	{attribute 'TcHmiSymbol.Show'}

	bSimulated:		BOOL;				// Flag indicating if the value is simulated.
	{attribute 'TcHmiSymbol.Show'}

	lrSimTempK:	LREAL;				// Simulated Temp [K]

	{attribute 'TcHmiSymbol.Show'}

	bEnabled:		BOOL	:= FALSE;	// Flag indicating if the voter is enabled
    
	{attribute 'TcHmiSymbol.Show'}

	sDescription:	STRING;	// User description of the voter (e.g. 'Average detector T')
    
	{attribute 'TcHmiSymbol.Show'}

	bValid:			BOOL	:= FALSE;	// Flag indicating if the value is valid.
	{attribute 'TcHmiSymbol.Show'}
	{attribute 'TcHmiSymbol.ReadOnly'}
	lrTempK:		LREAL;				// Calculated Temperature in K
	sStatus:		STRING;				// Status string

	// Flags indicating connected sensor is Valid.
	{attribute 'TcHmiSymbol.Show'}
	{attribute 'TcHmiSymbol.ReadOnly'}
	lrSens1TempK:		LREAL;
	{attribute 'TcHmiSymbol.Show'}
	{attribute 'TcHmiSymbol.ReadOnly'}
	lrSens2TempK:		LREAL;
	{attribute 'TcHmiSymbol.Show'}
	{attribute 'TcHmiSymbol.ReadOnly'}
	lrSens3TempK:		LREAL;
	{attribute 'TcHmiSymbol.Show'}
	{attribute 'TcHmiSymbol.ReadOnly'}
	lrSens4TempK:		LREAL;
	{attribute 'TcHmiSymbol.Show'}
	{attribute 'TcHmiSymbol.ReadOnly'}
	lrSens5TempK:		LREAL;
	
	{attribute 'TcHmiSymbol.Show'}
	{attribute 'TcHmiSymbol.ReadOnly'}
	bValidSensor1:		BOOL	:= FALSE;
	{attribute 'TcHmiSymbol.Show'}
	{attribute 'TcHmiSymbol.ReadOnly'}
	bValidSensor2:		BOOL	:= FALSE;
	{attribute 'TcHmiSymbol.Show'}
	{attribute 'TcHmiSymbol.ReadOnly'}
	bValidSensor3:		BOOL	:= FALSE;
	{attribute 'TcHmiSymbol.Show'}
	{attribute 'TcHmiSymbol.ReadOnly'}
	bValidSensor4:		BOOL	:= FALSE;
	{attribute 'TcHmiSymbol.Show'}
	{attribute 'TcHmiSymbol.ReadOnly'}
	bValidSensor5:		BOOL	:= FALSE;
	{attribute 'TcHmiSymbol.ShowRecursively'}

	stAlarms:		T_CRYO_ALARMS;	

	bInRange:		BOOL	:= FALSE;

	lrTempC:		LREAL;				// Temp [deg C]
	
	{attribute 'TcHmiSymbol.Show'}
	aTempIndexes:		ARRAY[0..4] OF E_ALL_METIS_TEMPERATURES;
	{attribute 'TcHmiSymbol.Show'}
	nVoteMethod:		E_METIS_TEMP_VOTE_METHOD;

    //bEnabled:       BOOL;	

END_STRUCT
END_TYPE

// DUTs/Structures/Temp_Voter/T_METIS_TEMP_VOTE_CFG
TYPE T_METIS_TEMP_VOTE_CFG :
STRUCT
    bEnabled        : BOOL;
    sDescription    : STRING; 

	sTemp1_Name	    : STRING;
	sTemp2_Name	    : STRING;
	sTemp3_Name	    : STRING;
	sTemp4_Name	    : STRING;
	sTemp5_Name	    : STRING;
	
	nVote_Method    : E_METIS_TEMP_VOTE_METHOD;
	
	eTemperature1   : E_ALL_METIS_TEMPERATURES;
	eTemperature2   : E_ALL_METIS_TEMPERATURES;
	eTemperature3   : E_ALL_METIS_TEMPERATURES;
	eTemperature4   : E_ALL_METIS_TEMPERATURES;
	eTemperature5   : E_ALL_METIS_TEMPERATURES;
	
END_STRUCT
END_TYPE

// DUTs/Structures/Temp_Voter/T_METIS_TEMP_VOTERS_CTRL
TYPE T_METIS_TEMP_VOTERS_CTRL :
STRUCT
	
	// CRY

    tor_vote_cry_1  :			FB_CRYO_CMD_OVERRIDE;
    tor_vote_cry_2  :           FB_CRYO_CMD_OVERRIDE;
    tor_vote_cry_3  :           FB_CRYO_CMD_OVERRIDE;
    tor_vote_cry_4  :           FB_CRYO_CMD_OVERRIDE;
    tor_vote_cry_5  :           FB_CRYO_CMD_OVERRIDE;
    tor_vote_cry_6  :           FB_CRYO_CMD_OVERRIDE;
    tor_vote_cry_7  :           FB_CRYO_CMD_OVERRIDE;
    tor_vote_cry_8  :           FB_CRYO_CMD_OVERRIDE;
    tor_vote_cry_9  :           FB_CRYO_CMD_OVERRIDE;
    tor_vote_cry_10 :           FB_CRYO_CMD_OVERRIDE;
                                
    // SCA                      
    tor_vote_sca_1  :           FB_CRYO_CMD_OVERRIDE;
    tor_vote_sca_2  :           FB_CRYO_CMD_OVERRIDE;
    tor_vote_sca_3  :           FB_CRYO_CMD_OVERRIDE;
    tor_vote_sca_4  :           FB_CRYO_CMD_OVERRIDE;
    tor_vote_sca_5  :           FB_CRYO_CMD_OVERRIDE;
    tor_vote_sca_6  :           FB_CRYO_CMD_OVERRIDE;
    tor_vote_sca_7  :           FB_CRYO_CMD_OVERRIDE;
    tor_vote_sca_8  :           FB_CRYO_CMD_OVERRIDE;
    tor_vote_sca_9  :           FB_CRYO_CMD_OVERRIDE;
    tor_vote_sca_10 :           FB_CRYO_CMD_OVERRIDE;
                                
    // IMG                      
    tor_vote_img_1  :           FB_CRYO_CMD_OVERRIDE;
    tor_vote_img_2  :           FB_CRYO_CMD_OVERRIDE;
    tor_vote_img_3  :           FB_CRYO_CMD_OVERRIDE;
    tor_vote_img_4  :           FB_CRYO_CMD_OVERRIDE;
    tor_vote_img_5  :           FB_CRYO_CMD_OVERRIDE;
    tor_vote_img_6  :           FB_CRYO_CMD_OVERRIDE;
    tor_vote_img_7  :           FB_CRYO_CMD_OVERRIDE;
    tor_vote_img_8  :           FB_CRYO_CMD_OVERRIDE;
    tor_vote_img_9  :           FB_CRYO_CMD_OVERRIDE;
    tor_vote_img_10 :           FB_CRYO_CMD_OVERRIDE;
                                
    // System temp               
    tor_vote_master_temp:       FB_CRYO_CMD_OVERRIDE;
    tor_vote_master_1   :       FB_CRYO_CMD_OVERRIDE;
    tor_vote_master_2   :       FB_CRYO_CMD_OVERRIDE;
	
	
// Temp Simulation Flag

	//CRY
	bSim_Temp_vote_cry_1  :		BOOL := FALSE;
    bSim_Temp_vote_cry_2  :     BOOL := FALSE;
    bSim_Temp_vote_cry_3  :     BOOL := FALSE;
    bSim_Temp_vote_cry_4  :     BOOL := FALSE;
    bSim_Temp_vote_cry_5  :     BOOL := FALSE;
    bSim_Temp_vote_cry_6  :     BOOL := FALSE;
    bSim_Temp_vote_cry_7  :     BOOL := FALSE;
    bSim_Temp_vote_cry_8  :     BOOL := FALSE;
    bSim_Temp_vote_cry_9  :     BOOL := FALSE;
    bSim_Temp_vote_cry_10 :     BOOL := FALSE;
                                
    //SCA                       
    bSim_Temp_vote_sca_1  :     BOOL := FALSE;
    bSim_Temp_vote_sca_2  :     BOOL := FALSE;
    bSim_Temp_vote_sca_3  :     BOOL := FALSE;
    bSim_Temp_vote_sca_4  :     BOOL := FALSE;
    bSim_Temp_vote_sca_5  :     BOOL := FALSE;
    bSim_Temp_vote_sca_6  :     BOOL := FALSE;
    bSim_Temp_vote_sca_7  :     BOOL := FALSE;
    bSim_Temp_vote_sca_8  :     BOOL := FALSE;
    bSim_Temp_vote_sca_9  :     BOOL := FALSE;
    bSim_Temp_vote_sca_10 :     BOOL := FALSE;
                                
	//IMG                       
    bSim_Temp_vote_img_1  :     BOOL := FALSE;
    bSim_Temp_vote_img_2  :     BOOL := FALSE;
    bSim_Temp_vote_img_3  :     BOOL := FALSE;
    bSim_Temp_vote_img_4  :     BOOL := FALSE;
    bSim_Temp_vote_img_5  :     BOOL := FALSE;
    bSim_Temp_vote_img_6  :     BOOL := FALSE;
    bSim_Temp_vote_img_7  :     BOOL := FALSE;
    bSim_Temp_vote_img_8  :     BOOL := FALSE;
    bSim_Temp_vote_img_9  :     BOOL := FALSE;
    bSim_Temp_vote_img_10 :     BOOL := FALSE;
                                
    //system temp               
    bSim_Temp_vote_master_temp: BOOL := FALSE;
    bSim_Temp_vote_master_1   : BOOL := FALSE;
    bSim_Temp_vote_master_2   : BOOL := FALSE;
                             
	
                               
END_STRUCT
END_TYPE

// DUTs/Structures/Temperature/E_ALL_METIS_TEMPERATURES
{attribute 'qualified_only'}
{attribute 'strict'}
{attribute 'to_string'}
TYPE E_ALL_METIS_TEMPERATURES :
(
	empty_temp 		:= 0,					
	(*Temp Cryo: 23 + 10 = 33 *)
	t_cry_sha_1		:= 1,			
	t_cry_sha_2		:= 2,			
	t_cry_sha_3		:= 3,			
	t_cry_sha_4		:= 4,           	
	t_cry_shb_1		:= 5,			
	t_cry_shb_2		:= 6,           	
	t_cry_shb_3		:= 7,           	
	t_cry_shb_4		:= 8,           	
	t_cry_shc_1		:= 9,			
	t_cry_shc_2		:= 10,           	
	t_cry_shc_3     := 11,           	
	t_cry_shc_4     := 12,           	
	t_cry_pta_1     := 13,           	
	t_cry_pta_2     := 14,           	
	t_cry_ptb_1     := 15,           	
	t_cry_ptb_2     := 16,           	
	t_cry_ptc_1		:= 17,			
	t_cry_ptc_2     := 18,           	
	t_cry_pta_3     := 19,           	
	t_cry_ptb_3     := 20,           	
	t_cry_ptc_3     := 21,           	
	t_cry_sp_1		:= 22,			
	t_cry_sp_2		:= 23,			
	// voter outputs (10)           
	t_cry_vot_1     := 24,            
	t_cry_vot_2     := 25,            
	t_cry_vot_3     := 26,            
	t_cry_vot_4     := 27,            
	t_cry_vot_5     := 28,            
	t_cry_vot_6     := 29,            
	t_cry_vot_7     := 30,            
	t_cry_vot_8     := 31,            
	t_cry_vot_9     := 32,            
	t_cry_vot_10    := 33,            
	                            
	(*SCA Temps: 16 + 4 + 10 + 3 = 33 *)  
	         
	// cu X2
	t_sca_fw_1       := 34,           
	t_sca_fw_2       := 35,           
	t_sca_lu_1       := 36,           
	t_sca_fm         := 37,           
	t_sca_fs         := 38,           
	t_sca_lu_2       := 39,           
	t_sca_mod        := 40,           
	t_sca_pyr		 := 41,		
	// cu X3                    
	t_sca_h_1        := 42,           
	t_sca_if_1       := 43,           
	t_sca_if_2       := 44,           
	t_sca_lu_3       := 45,           
	t_sca_bp_1       := 46,           
	t_sca_bp_2       := 47,           
	t_sca_bp_3       := 48,           
	t_sca_h_2        := 49,           
	// detector (4)             
	t_sca_det_1      := 50,           
	t_sca_det_2      := 51,           
	t_sca_dhs_1      := 52,           
	t_sca_dhs_2      := 53,           
// voter outputs(10)        
	t_sca_vot_1       := 54,          
	t_sca_vot_2       := 55,          
	t_sca_vot_3       := 56,          
	t_sca_vot_4       := 57,          
	t_sca_vot_5       := 58,          
	t_sca_vot_6       := 59,          
	t_sca_vot_7       := 60,          
	t_sca_vot_8       := 61,          
	t_sca_vot_9       := 62,          
	t_sca_vot_10      := 63,          
	// temperature controller ramps (3)
	t_sca_wuh_ramp    := 64,         
	t_sca_det_2_ramp  := 65,         
	t_sca_dhs_2_ramp  := 66,         
	
	(*IMG Temps : 24 + 6 + 10 + 4 = 44 *)              
	
	// cu (24)			  
	t_img_lpw_1        := 67,        
	t_img_lpw_2        := 68,         
	t_img_lfw_1        := 69,         
	t_img_lfw_2        := 70,         
	t_img_lpr_1        := 71,         
	t_img_bwu_3        := 72,         
	t_img_lnd_1        := 73,         
	t_img_lnd_2        := 74,         
	t_img_npw_1        := 75,         
	t_img_npw_2        := 76,         
	t_img_nfw_1        := 77,         
	t_img_nfw_2        := 78,         
	t_img_npr_1        := 79,         
	t_img_bwu_2        := 80,         
	t_img_nnd_1        := 81,         
	t_img_nnd_2        := 82,         
	t_img_opt_1        := 83,         
	t_img_bwu_1        := 84,         
	t_img_ctr_1        := 85,         
	t_img_ctr_2        := 86,         
	t_img_70k_1        := 87,         
	t_img_ln2_1        := 88,         
	t_img_ln2_2		   := 89,    
	t_img_hex_1        := 90,         
	// detector (6)             
	t_img_lmd_1        := 91,         
	t_img_lmd_2        := 92,         
	t_img_lmp_1        := 93,         
	t_img_lmp_2        := 94,         
	t_img_nd_1         := 95,         
	t_img_nd_2         := 96,         
	// voter outputs (10) 
	t_img_vot_1        := 97,      
	t_img_vot_2        := 98,        
	t_img_vot_3        := 99,       
	t_img_vot_4        := 100,       
	t_img_vot_5        := 101,       
	t_img_vot_6        := 102,       
	t_img_vot_7        := 103,       
	t_img_vot_8        := 104,       
	t_img_vot_9        := 105,       
	t_img_vot_10       := 106,       
// temperature controller       ramps (4)
	t_img_wuh_ramp     := 107,       
	t_img_lmd_2_ramp   := 108,       
	t_img_lmp_2_ramp   := 109,       
	t_img_nd_2_ramp    := 110,       
	                            
	(*Temp LMS : 16 *)          
	                            
	t_lms_pma_1        := 111,         
	t_lms_pma_2        := 112,         
	t_lms_msa_1        := 113,         
	t_lms_msa_2        := 114,         
	t_lms_pra_1        := 115,         
	t_lms_pra_2        := 116,         
	t_lms_gra_1        := 117,         
	t_lms_gra_2        := 118,         
	t_lms_pla_1        := 119,         
	t_lms_pla_2        := 120,         
	t_lms_pla_3        := 121,         
	t_lms_pla_4        := 122,         
	t_lms_tma          := 123,         
	t_lms_dtw          := 124,         
	t_lms_ptw          := 125,         
	t_lms_spare        := 126,         
	                            
	(*Temp CFO*) 
	
	
	// RTD temperatures   
	t_cry_pca          := 127,          // PCA.T = IMG Heat Exchanger Out
	t_cry_pcb          := 128,          // PCB.T = CFO Heat Exchanger Out
	t_cry_wim          := 129,          // WI.MT = Window Mount
	t_cry_wia          := 130,          // WI.AT = Window Ambient
                          
	// dew point temperatures
	t_cry_wid          := 131,         
	
	(*System temperatures   (3) *)
	// Master temperature to estimate overall temperature of the cryostat  
						  
	t_master           := 132,      	
	t_master_vot_1     := 133,      	
	t_master_vot_2     := 134     	
	                      

	
);
END_TYPE

// DUTs/Structures/Temperature/T_METIS_TEMPERATURE_STATUS
TYPE T_METIS_TEMPERATURE_STATUS EXTENDS T_METIS_SENSOR_BASE_STATUS:
STRUCT
	{attribute 'TcHmiSymbol.Show'}
    lrTempC : LREAL;
	{attribute 'TcHmiSymbol.Show'}
    lrTempK : LREAL;
END_STRUCT
END_TYPE

// HMI/DUTs/Cryo_Devices/Temperatures/E_HMI_TEMP_TABS
{attribute 'qualified_only'}
{attribute 'strict'}
TYPE E_HMI_TEMP_TABS :
(
    VOTERS
);
END_TYPE

// HMI/DUTs/Cryo_Devices/E_HMI_PUMPS_TABS
{attribute 'qualified_only'}
{attribute 'strict'}
TYPE E_HMI_PUMPS_TABS :
(
	RP_BRANCH_A := 0,
	TP_BRANCH_A,
	RP_BRANCH_B,
	TP_BRANCH_B
);
END_TYPE

// HMI/DUTs/Subsystems/CFO/E_HMI_CFO_TABS
{attribute 'qualified_only'}
{attribute 'strict'}
TYPE E_HMI_CFO_TABS :
(
	TEMPERATURES,
    VOTERS,
    HEATERS,
    TCONTROL
);
END_TYPE

// HMI/DUTs/Subsystems/CRY/Components/E_HMI_CRY_HEATER_TABS
{attribute 'qualified_only'}
{attribute 'strict'}
TYPE E_HMI_CRY_HEATER_TABS :
(
    H_CRY_SHA,
    H_CRY_SHB,
    H_CRY_SHC,
    H_CRY_SP,
    H_CRY_PTA,
    H_CRY_PTB,
    H_CRY_PTC,
    H_CRY_WI
);
END_TYPE

// HMI/DUTs/Subsystems/CRY/Components/E_HMI_CRY_TC_TABS
{attribute 'qualified_only'}
{attribute 'strict'}
TYPE E_HMI_CRY_TC_TABS :
(
	TC_CRY_SHA,
    TC_CRY_SHB,
    TC_CRY_SHC,
    TC_CRY_PT,
    TC_CRY_WI,
	TC_CRY_SP
);
END_TYPE

// HMI/DUTs/Subsystems/CRY/E_HMI_CRY_TABS
{attribute 'qualified_only'}
{attribute 'strict'}
TYPE E_HMI_CRY_TABS :
(
	TEMPERATURES,
    RH,
    HEATERS,
    VOTERS,
    TCONTROL,
	LN2CONTROL
);
END_TYPE

// HMI/DUTs/Subsystems/ICS/E_HMI_ICS_TABS
{attribute 'qualified_only'}
{attribute 'strict'}
TYPE E_HMI_ICS_TABS :
(
	CCU_NS_1,
	CCU_NS_2,
	CCU_CONFIGS
);
END_TYPE

// HMI/DUTs/Subsystems/IMG/Components/E_HMI_IMG_HEATER_TABS
{attribute 'qualified_only'}
{attribute 'strict'}
TYPE E_HMI_IMG_HEATER_TABS :
(
	H_IMG_WUH_1,
    H_IMG_WUH_2,
    H_IMG_LMD_2,
    H_IMG_LMP_2,
    H_IMG_ND_2
);
END_TYPE

// HMI/DUTs/Subsystems/IMG/Components/E_HMI_IMG_TC_TABS
{attribute 'qualified_only'}
{attribute 'strict'}
TYPE E_HMI_IMG_TC_TABS :
(
	TC_IMG_WUH,
    TC_IMG_LMD_2,
    TC_IMG_LMP_2,
    TC_IMG_ND_2
);
END_TYPE

// HMI/DUTs/Subsystems/IMG/E_HMI_IMG_TABS
{attribute 'qualified_only'}
{attribute 'strict'}
TYPE E_HMI_IMG_TABS :
(
	TEMPERATURES,
    VOTERS,
    TCONTROL,
    HEATERS,
    LAKESHORE_LM_DET,
    LAKESHORE_N_DET
);
END_TYPE

// HMI/DUTs/Subsystems/LMS/E_HMI_LMS_TABS
{attribute 'qualified_only'}
{attribute 'strict'}
TYPE E_HMI_LMS_TABS :
(
	TEMPERATURES,
    VOTERS,
    HEATERS,
    TCONTROL
);
END_TYPE

// HMI/DUTs/Subsystems/SCA/Components/E_HMI_SCA_HEATER_TABS
{attribute 'qualified_only'}
{attribute 'strict'}
TYPE E_HMI_SCA_HEATER_TABS :
(
	H_SCA_WUH_1,
    H_SCA_WUH_2,
    H_SCA_DET_2,
    H_SCA_DHS_2
);
END_TYPE

// HMI/DUTs/Subsystems/SCA/Components/E_HMI_SCA_TC_TABS
{attribute 'qualified_only'}
{attribute 'strict'}
TYPE E_HMI_SCA_TC_TABS :
(
	TC_SCA_WUH,
    TC_SCA_DET_2,
    TC_SCA_DHS_2
);
END_TYPE

// HMI/DUTs/Subsystems/SCA/E_HMI_SCA_TABS
{attribute 'qualified_only'}
{attribute 'strict'}
TYPE E_HMI_SCA_TABS :
(
	TEMPERATURES,
    VOTERS,
    TCONTROL,
    HEATERS,
    LAKESHORE_DET
);
END_TYPE

// HMI/DUTs/System/E_HMI_TABS
{attribute 'qualified_only'}
{attribute 'strict'}
TYPE E_HMI_TABS :
(
	HOME,
    SERVICES,
	EVACUATION,
    COOL_DOWN,
	WARM_UP,
	VENTING,
	ANTI_FOGGING,
	REGENERATION,
	POWER_OUTAGE,
	CABINETS,
	VALVES,
	CONTROL_UNITS,
	SUBSYSTEMS_CRY,
    SUBSYSTEMS_CFO,
    SUBSYSTEMS_IMG,
    SUBSYSTEMS_LMS,
    SUBSYSTEMS_SCA,
    SUBSYSTEMS_ICS,
	HEATERS,
	EVENTS,
	PRESSURES,
	COOLERS,
	PUMPS,
	TEMPERATURES,
	ICS_INTERLOCKS,
	DETECTORS,
	CONTROL_LOOPS,
	SIMULATION
	
);
END_TYPE

// HMI/DUTs/Util/E_HMI_COLORS
TYPE E_HMI_COLORS :
(
	GREEN := 16#FF00FF00,
	RED := 16#FFFF0000,
	ORANGE := 16#FFFF802D,
	GRAY := 16#FFD3D3D3,
	DARK_GRAY := 16#FF949494,
	BLACK := 16#FF000000,
	WHITE := 16#FFFFFFFF,
	BLUE := 16#FF0000FF
) DWORD;
END_TYPE

// HMI/DUTs/Util/E_HMI_VOTER_TABS
{attribute 'qualified_only'}
{attribute 'strict'}
TYPE E_HMI_VOTER_TABS :
(
	VOTER_1,
    VOTER_2,
    VOTER_3,
    VOTER_4,
    VOTER_5,
    VOTER_6,
    VOTER_7,
    VOTER_8,
    VOTER_9,
    VOTER_10
);
END_TYPE

// HMI/DUTs/Util/T_ECAT_MODULE
TYPE T_ECAT_MODULE :
STRUCT
    sName : STRING(32);
    sType : STRING(16);
    nState : UINT;
    sState : STRING(16);
    bError : BOOL;
    bDisabled : BOOL;
    bNotPresent : BOOL;
END_STRUCT
END_TYPE

// HMI/DUTs/Util/T_HMI_COLORS
TYPE T_HMI_COLORS :
STRUCT
    fg : E_HMI_COLORS; // foreground
    bg : E_HMI_COLORS; // background
END_STRUCT
END_TYPE

// POUs/Devices/DigitalOutput/T_METIS_DO_CTRL
TYPE T_METIS_DO_CTRL :
STRUCT
    bEnable : BOOL;
END_STRUCT
END_TYPE

// POUs/Devices/DigitalOutput/T_METIS_DO_STAT
TYPE T_METIS_DO_STAT :
STRUCT    
    bActive             : BOOL; // Actual output (TRUE = Active, FALSE = Inactie)
    
    bError              : BOOL; // summary of the fault flags
    
	bOvertemperature    : BOOL; // Over temperature fault
	bOpenLoad           : BOOL; // Open load fault
	bOverCurrent        : BOOL; // Over current fault
	bShortCircuit       : BOOL; // Short circuit fault
    
    sStatus             : STRING;
END_STRUCT
END_TYPE

// POUs/Devices/RH_Sensor/T_METIS_RH_SENSOR_STAT
TYPE T_METIS_RH_SENSOR_STAT EXTENDS T_CRYO_SENSOR_STATUS:
STRUCT
    lrRhFraction        : LREAL; // Relative Humidity as a fraction [0..1]
    lrRhPercent         : LREAL; // Relative Humidity as a percentage [0..100]
    lrDewPointTempC     : LREAL; // Dew point temperature in °C
    bDewPointTempValid  : BOOL;  // TRUE if the dew point is valid
END_STRUCT
END_TYPE

// HMI/POUs/Cryo-Routines/Anti-Fogging/FB_HMI_ANTI_FOGGING
FUNCTION_BLOCK FB_HMI_ANTI_FOGGING EXTENDS FB_HMI_COMPONENT
VAR_INPUT
END_VAR
VAR_OUTPUT
END_VAR
VAR
END_VAR
VAR_IN_OUT
	{attribute 'OPC.UA.DA' := '0'}
	fbInstance		: FB_METIS_CRYO_ANTI_FOGGING;
	{attribute 'OPC.UA.DA' := '0'}
	interlocks:						T_METIS_CRYO_INTERLOCKS;

END_VAR


fbHealthStatus( 
				bIsEnabled:= TRUE, 
				bIsGood := NOT fbInstance.stat.bError,
				bHasWarning := fbInstance.stat.bWarning OR interlocks.bInterlock_AntiFogging
				);
				
fbBusyStatus(
				bIsBusy := fbInstance.stat.bBusy,
				bIsEnabled := TRUE);
				
M_UpdateStatusColor();

END_FUNCTION_BLOCK

// HMI/POUs/Util/Component/FB_HMI_COMPONENT
FUNCTION_BLOCK FB_HMI_COMPONENT
VAR_INPUT
END_VAR
VAR_OUTPUT
    fbHealthStatus : FB_HMI_HEALTH_STATUS;
    fbBusyStatus : FB_HMI_BUSY_STATUS;
    fbStatusColor : T_HMI_COLORS;
END_VAR
VAR
END_VAR

METHOD PROTECTED M_UpdateStatusColor
VAR_INPUT
END_VAR
// health and busy states must be updated by the subtype before calling this method!
fbStatusColor := F_HMI_HEALTH_BUSY_TO_COLOR(fbHealthStatus, fbBusyStatus);
END_METHOD

END_FUNCTION_BLOCK

// HMI/POUs/Services/Status/FB_HMI_HEALTH_STATUS
FUNCTION_BLOCK FB_HMI_HEALTH_STATUS
VAR_INPUT
	// TRUE if the subject is in Good health
	bIsGood: BOOL;
	// TRUE to add a warning to the Good health state
	bHasWarning: BOOL := FALSE;
	// TRUE if the health status is used
	bIsEnabled: BOOL := TRUE;
END_VAR
VAR_OUTPUT
	// TRUE if the subject is enabled
	bEnabled: BOOL;
    // TRUE if the subject is in good health
	bGood: BOOL;
	// TRUE if the subject is in good health, but there are one or more warnings present
	bWarning: BOOL;
	// TRUE if the subject is in bad health
	bBad: BOOL;
END_VAR
VAR_IN_OUT
END_VAR
VAR
END_VAR

bEnabled := bIsEnabled;
bBad := (NOT(bIsGood)) AND bIsEnabled;
bGood := (bIsGood AND (NOT(bHasWarning))) AND bIsEnabled;
bWarning := (bIsGood AND bHasWarning) AND bIsEnabled;

END_FUNCTION_BLOCK

// HMI/POUs/Services/Status/FB_HMI_BUSY_STATUS
FUNCTION_BLOCK FB_HMI_BUSY_STATUS
VAR_INPUT
	// TRUE if busy
	bIsBusy: BOOL;
	// TRUE if the busy status is used
	bIsEnabled: BOOL := TRUE;
END_VAR
VAR_OUTPUT
	// TRUE if the subject is enabled
	bEnabled: BOOL;
	///The subject is idle
	bIdle: BOOL;
	///The subject is busy
	bBusy: BOOL;
END_VAR
VAR_IN_OUT
END_VAR
VAR
END_VAR

bBusy := bIsBusy AND bIsEnabled;
bIdle := (NOT(bIsBusy)) AND bIsEnabled;

END_FUNCTION_BLOCK

// HMI/POUs/Services/Status/F_HMI_HEALTH_BUSY_TO_COLOR
FUNCTION F_HMI_HEALTH_BUSY_TO_COLOR : T_HMI_COLORS
VAR_IN_OUT
    fbHealthStatus : FB_HMI_HEALTH_STATUS;
    fbBusyStatus   : FB_HMI_BUSY_STATUS;
END_VAR
VAR_OUTPUT
END_VAR
VAR
END_VAR

IF fbHealthStatus.bGood THEN
	IF fbBusyStatus.bBusy THEN
		F_HMI_HEALTH_BUSY_TO_COLOR.fg := E_HMI_COLORS.WHITE;
		F_HMI_HEALTH_BUSY_TO_COLOR.bg := E_HMI_COLORS.BLUE;
	ELSE
		F_HMI_HEALTH_BUSY_TO_COLOR.fg := E_HMI_COLORS.BLACK;
		F_HMI_HEALTH_BUSY_TO_COLOR.bg := E_HMI_COLORS.GREEN;
	END_IF
ELSIF fbHealthStatus.bBad THEN
	F_HMI_HEALTH_BUSY_TO_COLOR.fg := E_HMI_COLORS.WHITE;
	F_HMI_HEALTH_BUSY_TO_COLOR.bg := E_HMI_COLORS.RED;
ELSIF fbHealthStatus.bWarning THEN
	F_HMI_HEALTH_BUSY_TO_COLOR.fg := E_HMI_COLORS.WHITE;
	F_HMI_HEALTH_BUSY_TO_COLOR.bg := E_HMI_COLORS.ORANGE;
ELSE
	F_HMI_HEALTH_BUSY_TO_COLOR.fg := E_HMI_COLORS.BLACK;
	F_HMI_HEALTH_BUSY_TO_COLOR.bg := E_HMI_COLORS.GRAY;
END_IF

END_FUNCTION

// POUs/Routines/AntiFogging/FB_METIS_CRYO_ANTI_FOGGING
FUNCTION_BLOCK FB_METIS_CRYO_ANTI_FOGGING
VAR_INPUT
	in_sName:							STRING := 'ANTI-FOGGING';
	in_bEnable:							BOOL := FALSE;
	in_Cryo_Stat:						T_METIS_CRYO_STAT;
	in_lrAntiFog_Purging_DewPoint:		LREAL := 10.0; // If dew-point is <10 K below ambient window purging is started
	in_lrAntiFog_Heating_DewPoint:		LREAL := 10.0; // If dew-point is <5 K below ambient window increased window heating is started
	in_lrAntiFog_DewPoint_Alarm:		LREAL := 5.0;  // dew point is <5 K below window temperature
END_VAR
VAR_OUTPUT
	out_bAntiFoggingActive:			BOOL := FALSE;
END_VAR
VAR_IN_OUT
	{attribute 'OPC.UA.DA' := '0'}
	all_cryo_temps:					FB_METIS_TEMPERATURES;
	{attribute 'OPC.UA.DA' := '0'}
	all_heaters:					FB_METIS_HEATERS;
	{attribute 'OPC.UA.DA' := '0'}
	all_t_ctrls:      				FB_METIS_TCTRL;
	{attribute 'OPC.UA.DA' := '0'}
	all_t_votes: 					FB_METIS_VOTERS;
	{attribute 'OPC.UA.DA' := '0'}
	interlocks:						T_METIS_CRYO_INTERLOCKS;
END_VAR
VAR
	stat:						T_MET_CRYO_ANTI_FOGGING_STAT;
	ctrl:						T_MET_CRYO_ANTI_FOGGING_CTRL;
	{attribute 'TcHmiSymbol.Show'}
	dryair_blow_valve: FB_METIS_CONTROL_VALVE;
	
	/////////////////////
	// Cryo System logs
	/////////////////////
		
	logs:	FB_CRYO_FUNCTION_LOG;	
	
			//
	// Triggers.
	//
	// Capture Enable/Disable.
	trigEnable:		R_TRIG;	// in_bEnable
	trigDisable:	F_TRIG;	// in_bEnable
	
END_VAR
VAR CONSTANT

    // --- [5000] Preconditions ---
    E5000_CryostatIsWarm                          : UDINT := 5000001; // Anti-fogging requested while cryostat is warm
    E5001_CryostatNotInVacuum                     : UDINT := 5000002; // Cryostat is not under vacuum
    E5002_DewPointNotSufficientlyBelowAmbient     : UDINT := 5000003; // Dew point is not at least 10 K below ambient at start
    E5003_AntiFoggingAlreadyActive                : UDINT := 5000004; // Anti-fogging requested while already active
    E5004_AmbientTemperatureSensorFault           : UDINT := 5000005; // Ambient temperature sensor invalid or faulty
    E5005_DewPointSensorFault                     : UDINT := 5000006; // Dew-point sensor invalid or faulty
    E5006_WindowTemperatureSensorFault            : UDINT := 5000007; // Window or window flange temperature sensor invalid or faulty

    // --- [5100] Heater / Blower / Actuator Errors ---
    E5100_WindowFlangeControlFailedToStart        : UDINT := 5100001; // Window flange temperature control failed to start
    E5101_WindowHeaterFailure                     : UDINT := 5100002; // Window heater failed or not responding
    E5102_PurgeBlowerFailedToStart                : UDINT := 5100003; // Dry air / nitrogen blower failed to start
    E5103_PurgeFlowControlFault                   : UDINT := 5100004; // Purge flow control failed or unstable
    E5104_WindowHeaterFailedToIncreaseOutput      : UDINT := 5100005; // Increased window heating could not be applied
    E5105_BlowerFailedToReachMaximum              : UDINT := 5100006; // Blower failed to reach maximum demand during alarm action
    E5106_AntiFoggingActuatorShutdownFailure      : UDINT := 5100007; // Heater or blower failed to stop during shutdown

    // --- [5200] Dew Point / Temperature Monitoring Errors ---
    E5200_DewPointTooCloseToAmbient               : UDINT := 5200001; // Dew point is less than 10 K below ambient
    E5201_DewPointTooCloseToWindowTemperature     : UDINT := 5200002; // Dew point is less than 10 K below window temperature
    E5202_DewPointCriticalMargin                  : UDINT := 5200003; // Dew point is less than 5 K below ambient
    E5203_WindowCondensationRiskHigh              : UDINT := 5200004; // Dew point is less than 5 K below window temperature
    E5204_WindowTemperatureTooLow                 : UDINT := 5200005; // Window temperature too low for current dew point conditions
    E5205_WindowFlangeControlDeviation            : UDINT := 5200006; // Window flange temperature deviates excessively from setpoint
    E5206_DewPointNotImprovingDuringPurging       : UDINT := 5200007; // Dew point did not improve after purge started
    E5207_DewPointNotImprovingDuringHeating       : UDINT := 5200008; // Dew point margin did not improve after increased heating started

    // --- [5300] Sequence Timing Errors ---
    E5300_PurgeStartTimeout                       : UDINT := 5300001; // Purging did not start within allowed time
    E5301_HeatingBoostStartTimeout                : UDINT := 5300002; // Increased window heating did not start within allowed time
    E5302_DewPointRecoveryTimeout                 : UDINT := 5300003; // Dew point margin did not recover within allowed time
    E5303_AntiFoggingSequenceTimeout              : UDINT := 5300004; // Anti-fogging sequence exceeded maximum allowed duration

    // --- [5400] Manual Intervention / Abort ---
    E5400_OperatorAbortedAntiFogging              : UDINT := 5400001; // Operator manually stopped anti-fogging
    E5401_OperatorDisabledWindowHeating           : UDINT := 5400002; // Operator manually disabled window heating
    E5402_OperatorDisabledPurging                 : UDINT := 5400003; // Operator manually disabled purge flow
    E5403_OperatorChangedAntiFoggingMode          : UDINT := 5400004; // Operator changed anti-fogging mode unexpectedly

    // --- [5500] Interlock Violations ---
    E5500_AntiFoggingActiveWhileCryostatWarm      : UDINT := 5500001; // Anti-fogging remained active although cryostat is warm
    E5501_AntiFoggingActiveWithoutVacuum          : UDINT := 5500002; // Anti-fogging active while cryostat is not under vacuum
    E5502_PurgeRequestedWithoutValidDewPoint      : UDINT := 5500003; // Purging requested without valid dew-point measurement
    E5503_HeatingBoostRequestedWithoutValidTemps  : UDINT := 5500004; // Heating boost requested without valid temperature inputs

    // --- [5600] Alarm / Protective Action Failures ---
    E5600_AlarmAction_HeatingNotApplied           : UDINT := 5600001; // Heating to 10 K above ambient could not be applied during alarm
    E5601_AlarmAction_BlowerNotAtMaximum          : UDINT := 5600002; // Blower could not be driven to maximum during alarm
    E5602_CondensationProtectionNotAchieved       : UDINT := 5600003; // Required condensation protection margin could not be achieved

END_VAR


IF stat.bAuto THEN
	ctrl.bEnable := in_bEnable;
ELSE
	;
END_IF

M_HandleEvents();

M_StateMachine(			all_cryo_temps:= all_cryo_temps,
						all_heaters := all_heaters,
						all_t_ctrls := all_t_ctrls,
						all_t_votes := all_t_votes,
						interlocks := interlocks);

M_ExecuteControllers();

M_UpdateStatus(			all_cryo_temps:= all_cryo_temps,
						all_heaters := all_heaters,
						all_t_ctrls := all_t_ctrls,
						all_t_votes := all_t_votes,
						interlocks := interlocks);

METHOD M_Activity_AirBlowing : BOOL
VAR_INPUT
END_VAR
VAR_IN_OUT
	{attribute 'OPC.UA.DA' := '0'}
	all_cryo_temps:					FB_METIS_TEMPERATURES;
	{attribute 'OPC.UA.DA' := '0'}
	all_heaters:					FB_METIS_HEATERS;
	{attribute 'OPC.UA.DA' := '0'}
	all_t_ctrls:      				FB_METIS_TCTRL;
	{attribute 'OPC.UA.DA' := '0'}
	all_t_votes: 					FB_METIS_VOTERS;
	{attribute 'OPC.UA.DA' := '0'}
	interlocks:						T_METIS_CRYO_INTERLOCKS;
END_VAR
VAR_INST
    nAirBlowingSubState : INT := 0;
    nextState           : E_MET_CRYO_ANTI_FOGGING_STATE;
END_VAR
CASE nAirBlowingSubState OF


    0: // Initialization step

	
		// Starting Blower
        IF dryair_blow_valve.stat.bError THEN
            logs.M_LogWarning('Anti-Fogging: Air blower valve fault. Transitioning to ERROR state.');
            stat.nState := E_MET_CRYO_ANTI_FOGGING_STATE.ERROR;
            RETURN;
        END_IF

        IF dryair_blow_valve.stat.bActive THEN
            dryair_blow_valve.M_Activity_Valve_Normal();
            logs.M_LogInfo('Anti-Fogging: Dry air purge activated.');
        END_IF

        // Optional: Control output flow via PID or HMI — future enhancement

		// Starting heater if not active already
		 IF NOT all_heaters.h_cry_wi.M_isHeaterInError() THEN
            IF NOT all_heaters.h_cry_wi.stat.bActive THEN
                all_heaters.h_cry_wi.M_SetEnable();
                logs.M_LogInfo('Anti-Fogging: Shield heater enabled for standard operation.');
            END_IF

            IF NOT all_t_ctrls.tc_cry_wi.stat.bStarted THEN
                all_t_ctrls.tc_cry_wi.M_SetEnable();
                logs.M_LogInfo('Anti-Fogging: Temperature control enabled for window mount.');
            END_IF

            // Set ambient control point
            all_t_ctrls.tc_cry_wi.M_Set_SetPoint(
                m_eSetpointType := E_METIS_CTRL_SETPOINT_SWITCH.FIXED,
                m_lrFixedSetpoint := in_Cryo_Stat.lrAmbiantTempC,
                m_lrSetpointOffset := 1.0,
                m_pSetpointTemp := all_cryo_temps.M_SetTemperatureSensor(0));

            logs.M_LogInfo('Anti-Fogging: Setpoint adjusted to ambient tracking for window flange.');
        ELSE
            logs.M_LogWarning('Anti-Fogging: Heater error detected. Switching to ERROR state.');
            stat.nState := E_MET_CRYO_ANTI_FOGGING_STATE.ERROR;
            RETURN;
        END_IF		
		
		

        nAirBlowingSubState := 10;
        RETURN;


    10: // Monitoring and evaluation

		M_Evaluate_DewPoint_State(nNextState => nextState);
		
        IF nextState <> E_MET_CRYO_ANTI_FOGGING_STATE.AIR_BLOWING THEN
            stat.nState := nextState;
            nAirBlowingSubState := 0; // Reset internal state
        END_IF
        RETURN;

END_CASE
END_METHOD

METHOD M_Activity_Alarm_Condition : BOOL
VAR_INPUT
END_VAR
VAR_IN_OUT
	{attribute 'OPC.UA.DA' := '0'}
	all_cryo_temps:					FB_METIS_TEMPERATURES;
	{attribute 'OPC.UA.DA' := '0'}
	all_heaters:					FB_METIS_HEATERS;
	{attribute 'OPC.UA.DA' := '0'}
	all_t_ctrls:      				FB_METIS_TCTRL;
	{attribute 'OPC.UA.DA' := '0'}
	all_t_votes: 					FB_METIS_VOTERS;
	{attribute 'OPC.UA.DA' := '0'}
	interlocks:						T_METIS_CRYO_INTERLOCKS;
END_VAR
VAR_INST
    nAlarmSubState : INT := 0;
    nextState           : E_MET_CRYO_ANTI_FOGGING_STATE;
    sLogMsg             : STRING;
END_VAR

//IF dew point is <5 K below window temperature
//	o	Window heating 10 K above ambient
//	o	Dry air blower to maximum

CASE nAlarmSubState OF

	0: // Initialization
		// Check for heater error first
		IF all_heaters.h_cry_wi.M_isHeaterInError() THEN
			logs.M_LogWarning('Anti-Fogging: Heater error detected. Switching to ERROR state.');
			stat.nState := E_MET_CRYO_ANTI_FOGGING_STATE.ERROR;
			RETURN;
		END_IF

		// Enable heater if not already on
		IF NOT all_heaters.h_cry_wi.stat.bActive THEN
			all_heaters.h_cry_wi.M_SetEnable();
			logs.M_LogInfo('Anti-Fogging: Heater enabled for alarm condition.');
		END_IF

		// Enable temperature controller if not yet started
		IF NOT all_t_ctrls.tc_cry_wi.stat.bStarted THEN
			all_t_ctrls.tc_cry_wi.M_SetEnable();
			logs.M_LogInfo('Anti-Fogging: Temp controller enabled.');
		END_IF

		// Check blower
		IF dryair_blow_valve.stat.bError THEN
			logs.M_LogWarning('Anti-Fogging: Air valve error. Switching to ERROR state.');
			stat.nState := E_MET_CRYO_ANTI_FOGGING_STATE.ERROR;
			RETURN;
		END_IF

		// Activate blower if not already active
		IF NOT dryair_blow_valve.stat.bActive THEN
			dryair_blow_valve.M_SetEnable();
			logs.M_LogInfo('Anti-Fogging: Air purge started.');
		END_IF

		// Set blower to maximum
		dryair_blow_valve.M_Activity_Valve_Alarm();

		// Track ambient +10K using sensor t_cry_wia
		all_t_ctrls.tc_cry_wi.M_Set_SetPoint(
			m_eSetpointType := E_METIS_CTRL_SETPOINT_SWITCH.VARIABLE,
			m_lrFixedSetpoint := 0.0,
			m_lrSetpointOffset := 10.0,
			m_pSetpointTemp := all_cryo_temps.M_SetTemperatureSensor(
				m_nIndex := all_cryo_temps.M_GetTempSensorIndex('t_cry_wia'))
		);

		logs.M_LogInfo('Anti-Fogging: Heater setpoint = Ambient +10K.');
		nAlarmSubState := 10;
		RETURN;

	10: // Monitoring
		M_Evaluate_DewPoint_State(nNextState => nextState);

		IF nextState <> E_MET_CRYO_ANTI_FOGGING_STATE.ALARM_CONDITION THEN
			stat.nState := nextState;
			nAlarmSubState := 0;
		END_IF
		RETURN;

END_CASE
END_METHOD

METHOD M_Activity_Check_Preconditions
VAR_INPUT
END_VAR
VAR_IN_OUT
	{attribute 'OPC.UA.DA' := '0'}
	all_cryo_temps:					FB_METIS_TEMPERATURES;
	{attribute 'OPC.UA.DA' := '0'}
	all_heaters:					FB_METIS_HEATERS;
	{attribute 'OPC.UA.DA' := '0'}
	all_t_ctrls:      				FB_METIS_TCTRL;
	{attribute 'OPC.UA.DA' := '0'}
	all_t_votes: 					FB_METIS_VOTERS;
	{attribute 'OPC.UA.DA' := '0'}
	interlocks:						T_METIS_CRYO_INTERLOCKS;
END_VAR

stat.bActive := TRUE;


// Check core preconditions
IF in_Cryo_Stat.bInVacuum AND NOT in_Cryo_Stat.bWarm  THEN

    logs.M_LogInfo('Anti-Fogging preconditions met. Proceeding...');
	stat.sState := 'Anti-Fogging preconditions met. Proceeding...';
    stat.nState := E_MET_CRYO_ANTI_FOGGING_STATE.START_ANTI_FOGGING;

ELSE
    // If Cool Down has started, still allow Anti-Fogging to begin 
    IF in_Cryo_Stat.bCoolDownActive THEN
        logs.M_LogInfo('Cool Down is active. Forcing Anti-Fogging start...');
        stat.nState := E_MET_CRYO_ANTI_FOGGING_STATE.START_ANTI_FOGGING;
		
		stat.bActive := TRUE;
		stat.bDone := FALSE;
		stat.bBusy := TRUE;
    ELSE
        // Otherwise, raise error and wait
        stat.nState := E_MET_CRYO_ANTI_FOGGING_STATE.ERROR;
        stat.sState := 'Preconditions Not Satisfied for Anti-Fogging';
        //M_SetError(E2113_PreConditions_Failed, 'Anti-Fogging precondition check failed.');
    END_IF
END_IF
END_METHOD

METHOD M_Activity_Error_Handling
VAR_INPUT
END_VAR
VAR_IN_OUT
	{attribute 'OPC.UA.DA' := '0'}
	all_cryo_temps:					FB_METIS_TEMPERATURES;
	{attribute 'OPC.UA.DA' := '0'}
	all_heaters:					FB_METIS_HEATERS;
	{attribute 'OPC.UA.DA' := '0'}
	all_t_ctrls:      				FB_METIS_TCTRL;
	{attribute 'OPC.UA.DA' := '0'}
	all_t_votes: 					FB_METIS_VOTERS;
	{attribute 'OPC.UA.DA' := '0'}
	interlocks:						T_METIS_CRYO_INTERLOCKS;
END_VAR
stat.bError := TRUE;



IF ctrl.bReset THEN

	IF all_heaters.h_cry_wi.stat.bActive THEN
		all_heaters.h_cry_wi.M_SetDisable();
		logs.M_LogInfo('Anti-Fogging: Disabling window heater...');
	END_IF
	
	IF all_t_ctrls.tc_cry_wi.stat.bStarted THEN
		all_t_ctrls.tc_cry_wi.M_SetDisable();
		logs.M_LogInfo('Anti-Fogging: Disabling temperature controller...');
	END_IF
	
	IF dryair_blow_valve.stat.bActive THEN
		dryair_blow_valve.M_SetDisable();
		logs.M_LogInfo('Anti-Fogging: Disabling dry air blower...');
	END_IF
 
	stat.nState := E_MET_CRYO_ANTI_FOGGING_STATE.NONE;
	ctrl.bReset := FALSE;
	ctrl.bEnable := FALSE;
	stat.bError := FALSE;						
END_IF
END_METHOD

METHOD M_Activity_Finished : BOOL
VAR_INPUT
END_VAR
VAR_IN_OUT
	{attribute 'OPC.UA.DA' := '0'}
	all_cryo_temps:					FB_METIS_TEMPERATURES;
	{attribute 'OPC.UA.DA' := '0'}
	all_heaters:					FB_METIS_HEATERS;
	{attribute 'OPC.UA.DA' := '0'}
	all_t_ctrls:      				FB_METIS_TCTRL;
	{attribute 'OPC.UA.DA' := '0'}
	all_t_votes: 					FB_METIS_VOTERS;
	{attribute 'OPC.UA.DA' := '0'}
	interlocks:						T_METIS_CRYO_INTERLOCKS;
END_VAR
VAR_INST
    nRetryCounter : INT := 0;
    bAllOff       : BOOL := FALSE;
    nMaxRetries   : INT := 3;
END_VAR
// === Disable components ===
IF all_heaters.h_cry_wi.stat.bActive THEN
    all_heaters.h_cry_wi.M_SetDisable();
    logs.M_LogInfo('Anti-Fogging: Disabling window heater...');
END_IF

IF all_t_ctrls.tc_cry_wi.stat.bStarted THEN
    all_t_ctrls.tc_cry_wi.M_SetDisable();
    logs.M_LogInfo('Anti-Fogging: Disabling temperature controller...');
END_IF

//IF dryair_blow_valve.stat.bActive THEN
//    dryair_blow_valve.M_SetDisable();
//    logs.M_LogInfo('Anti-Fogging: Disabling dry air blower...');
//END_IF

// === Check shutdown status ===
bAllOff := NOT all_heaters.h_cry_wi.stat.bActive
           AND NOT all_t_ctrls.tc_cry_wi.stat.bStarted;
           //AND NOT dryair_blow_valve.stat.bActive;

IF bAllOff THEN
    logs.M_LogInfo('Anti-Fogging: All components successfully disabled.');
    stat.nState := E_MET_CRYO_ANTI_FOGGING_STATE.NONE;
    stat.sState := 'Anti-Fogging OFF';
		stat.bActive := FALSE;
		stat.bDone := TRUE;
		stat.bBusy := FALSE;
    RETURN;
ELSE
    nRetryCounter := nRetryCounter + 1;
    //logs.M_LogWarning('Anti-Fogging: Some components did not disable. Attempt #: ' + INT_TO_STRING(nRetryCounter));

    IF nRetryCounter >= nMaxRetries THEN
        logs.M_LogWarning('Anti-Fogging: Disabling Attempts Failed. Entering ERROR state.');
        stat.nState := E_MET_CRYO_ANTI_FOGGING_STATE.ERROR;
        stat.sState := 'Error: Shutdown Failure in Anti-Fogging';
        RETURN;
    ELSE
        // Allow retry on next cycle
        RETURN;
    END_IF
END_IF
END_METHOD

METHOD M_Activity_Heating : BOOL
VAR_INPUT
END_VAR
VAR_IN_OUT
	{attribute 'OPC.UA.DA' := '0'}
	all_cryo_temps:					FB_METIS_TEMPERATURES;
	{attribute 'OPC.UA.DA' := '0'}
	all_heaters:					FB_METIS_HEATERS;
	{attribute 'OPC.UA.DA' := '0'}
	all_t_ctrls:      				FB_METIS_TCTRL;
	{attribute 'OPC.UA.DA' := '0'}
	all_t_votes: 					FB_METIS_VOTERS;
	{attribute 'OPC.UA.DA' := '0'}
	interlocks:						T_METIS_CRYO_INTERLOCKS;
END_VAR
VAR_INST
    nHeatingSubState : INT := 0;
    nextState           : E_MET_CRYO_ANTI_FOGGING_STATE;
    sLogMsg             : STRING;
END_VAR
(*	If dew-point is <5 K below ambient window increased window heating is started
	o	flange is heated 10 K above dew point
*)

CASE nHeatingSubState OF


    0: // Initialization step

        IF NOT all_heaters.h_cry_wi.M_isHeaterInError() THEN
            IF NOT all_heaters.h_cry_wi.stat.bActive THEN
                all_heaters.h_cry_wi.M_SetEnable();
                logs.M_LogInfo('Anti-Fogging: Shield heater enabled for standard operation.');
            END_IF

            IF NOT all_t_ctrls.tc_cry_wi.stat.bStarted THEN
                all_t_ctrls.tc_cry_wi.M_SetEnable();
                logs.M_LogInfo('Anti-Fogging: Temperature control enabled for window mount.');
            END_IF

            // Set flange is heated 10 K above dew point
			
            all_t_ctrls.tc_cry_wi.M_Set_SetPoint(
                m_eSetpointType := E_METIS_CTRL_SETPOINT_SWITCH.FIXED,
                m_lrFixedSetpoint := in_Cryo_Stat.lrDewPointTempK + 10,
                m_lrSetpointOffset := 1.0,
                m_pSetpointTemp := all_cryo_temps.M_SetTemperatureSensor(0));

            logs.M_LogInfo('Anti-Fogging: Setpoint adjusted to heat flange 10 K above dew point');
            nHeatingSubState := 10; // Move to monitoring
        ELSE
            logs.M_LogWarning('Anti-Fogging: Heater error detected. Switching to ERROR state.');
            stat.nState := E_MET_CRYO_ANTI_FOGGING_STATE.ERROR;
            RETURN;
        END_IF
        RETURN;

    10: // Monitoring step
        // Evaluate dew point trends
		M_Evaluate_DewPoint_State(nNextState => nextState);
		
        IF nextState <> E_MET_CRYO_ANTI_FOGGING_STATE.HEATING THEN
            stat.nState := nextState;
            nHeatingSubState := 0; // Reset for next entry
        END_IF
        RETURN;

END_CASE
END_METHOD

METHOD M_Activity_None
VAR_INPUT
END_VAR
VAR_IN_OUT
	{attribute 'OPC.UA.DA' := '0'}
	all_cryo_temps:					FB_METIS_TEMPERATURES;
	{attribute 'OPC.UA.DA' := '0'}
	all_heaters:					FB_METIS_HEATERS;
	{attribute 'OPC.UA.DA' := '0'}
	all_t_ctrls:      				FB_METIS_TCTRL;
	{attribute 'OPC.UA.DA' := '0'}
	all_t_votes: 					FB_METIS_VOTERS;
	{attribute 'OPC.UA.DA' := '0'}
	interlocks:						T_METIS_CRYO_INTERLOCKS;
END_VAR
VAR
    nNextState : E_MET_CRYO_ANTI_FOGGING_STATE;
END_VAR
stat.bActive := FALSE;
stat.bDone := TRUE;
stat.bBusy := FALSE;


dryair_blow_valve.M_Activity_Valve_None();



// Check conditions for activation
IF NOT interlocks.bInterlock_AntiFogging THEN

    // If operator enabled anti-fogging, start as usual
    IF ctrl.bEnable THEN
        stat.nState := E_MET_CRYO_ANTI_FOGGING_STATE.CHECK_PRECONDITIONS;
        stat.sState := 'Anti-Fogging: Operator enabled, checking preconditions.';
        RETURN;
    END_IF

	IF in_Cryo_Stat.bInGoodVacuum OR in_Cryo_Stat.bInVacuum THEN
			// If cooling has started, auto-start antifogging based on dewpoint logic
			IF (in_Cryo_Stat.bCoolDownActive) OR (NOT in_Cryo_Stat.bWarm) THEN
				M_Evaluate_DewPoint_State(nNextState => nNextState);
		
				// Start antifogging automatically if needed
				IF nNextState <> E_MET_CRYO_ANTI_FOGGING_STATE.FINISHED THEN
					stat.nState := E_MET_CRYO_ANTI_FOGGING_STATE.CHECK_PRECONDITIONS;
					stat.sState := 'Anti-Fogging: Auto-start due to cooldown & humidity conditions.';
					RETURN;
				END_IF
			END_IF
	END_IF
END_IF

// Default: stay in NONE
stat.nState := E_MET_CRYO_ANTI_FOGGING_STATE.NONE;
stat.sState := 'Anti-Fogging OFF';
END_METHOD

METHOD M_Activity_Standard_Operation : BOOL
VAR_INPUT
END_VAR
VAR_IN_OUT
	{attribute 'OPC.UA.DA' := '0'}
	all_cryo_temps:					FB_METIS_TEMPERATURES;
	{attribute 'OPC.UA.DA' := '0'}
	all_heaters:					FB_METIS_HEATERS;
	{attribute 'OPC.UA.DA' := '0'}
	all_t_ctrls:      				FB_METIS_TCTRL;
	{attribute 'OPC.UA.DA' := '0'}
	all_t_votes: 					FB_METIS_VOTERS;
	{attribute 'OPC.UA.DA' := '0'}
	interlocks:						T_METIS_CRYO_INTERLOCKS;
END_VAR
VAR_INST
    nStandardOpSubState : INT := 0;
    nextState           : E_MET_CRYO_ANTI_FOGGING_STATE;
    sLogMsg             : STRING;
END_VAR
CASE nStandardOpSubState OF


    0: // Initialization step

        IF NOT all_heaters.h_cry_wi.M_isHeaterInError() THEN
            IF NOT all_heaters.h_cry_wi.stat.bActive THEN
                all_heaters.h_cry_wi.M_SetEnable();
                logs.M_LogInfo('Anti-Fogging: Shield heater enabled for standard operation.');
            END_IF

            IF NOT all_t_ctrls.tc_cry_wi.stat.bStarted THEN
                all_t_ctrls.tc_cry_wi.M_SetEnable();
                logs.M_LogInfo('Anti-Fogging: Temperature control enabled for window mount.');
            END_IF

            // Set ambient control point
            all_t_ctrls.tc_cry_wi.M_Set_SetPoint(
                m_eSetpointType := E_METIS_CTRL_SETPOINT_SWITCH.FIXED,
                m_lrFixedSetpoint := in_Cryo_Stat.lrAmbiantTempK,
                m_lrSetpointOffset := 1.0,
                m_pSetpointTemp := all_cryo_temps.M_SetTemperatureSensor(0));

            logs.M_LogInfo('Anti-Fogging: Setpoint adjusted to ambient tracking for window flange.');
            nStandardOpSubState := 10; // Move to monitoring
        ELSE
            logs.M_LogWarning('Anti-Fogging: Heater error detected. Switching to ERROR state.');
            stat.nState := E_MET_CRYO_ANTI_FOGGING_STATE.ERROR;
            RETURN;
        END_IF
        RETURN;

    10: // Monitoring step
        // Evaluate dew point trends
		M_Evaluate_DewPoint_State(nNextState => nextState);

        IF nextState <> E_MET_CRYO_ANTI_FOGGING_STATE.STANDARD_OPERATION THEN
            stat.nState := nextState;
            nStandardOpSubState := 0; // Reset for next entry
        END_IF
        RETURN;

END_CASE
END_METHOD

METHOD M_Activity_Start_Anti_Fogging : BOOL
VAR_INPUT
END_VAR
VAR_IN_OUT
	{attribute 'OPC.UA.DA' := '0'}
	all_cryo_temps:					FB_METIS_TEMPERATURES;
	{attribute 'OPC.UA.DA' := '0'}
	all_heaters:					FB_METIS_HEATERS;
	{attribute 'OPC.UA.DA' := '0'}
	all_t_ctrls:      				FB_METIS_TCTRL;
	{attribute 'OPC.UA.DA' := '0'}
	all_t_votes: 					FB_METIS_VOTERS;
	{attribute 'OPC.UA.DA' := '0'}
	interlocks:						T_METIS_CRYO_INTERLOCKS;
END_VAR
// Check for heater fault first
IF all_heaters.h_cry_wi.M_isHeaterInError() THEN
    logs.M_LogWarning('Anti-Fogging heater error detected.');
    //M_SetError(E2104_WindowHeaterError, 'Window heater error: Anti-fogging cannot proceed.');
    stat.nState := E_MET_CRYO_ANTI_FOGGING_STATE.ERROR;
    RETURN;
END_IF



M_Evaluate_DewPoint_State(nNextState => stat.nState);
END_METHOD

METHOD M_Configure
VAR_INPUT
END_VAR

IF NOT stat.bConfigured THEN
	

// This call just configures logs at the very start.
// Logging is done by explicit calls to M_LogInfo().
logs(in_sName := in_sName);


stat.bConfigured := TRUE;

END_IF
END_METHOD

METHOD PRIVATE M_Evaluate_DewPoint_State : BOOL
VAR_INPUT
END_VAR
VAR_OUTPUT
    nNextState: 	E_MET_CRYO_ANTI_FOGGING_STATE;
END_VAR
VAR
	prevState : E_MET_CRYO_ANTI_FOGGING_STATE;
END_VAR
prevState := stat.nState; 

IF NOT trigDisable.Q THEN

	// 1. Emergency stop condition: Cryostat is warm -> exit
	IF in_Cryo_Stat.bWarm THEN
		nNextState := E_MET_CRYO_ANTI_FOGGING_STATE.FINISHED;

	// 2. Alarm: dew point dangerously close to window temp
	ELSIF in_Cryo_Stat.lrDewPointTempC >= (in_Cryo_Stat.lrWindowMountTempC - 5.0) THEN
		nNextState := E_MET_CRYO_ANTI_FOGGING_STATE.ALARM_CONDITION;

	// 3. Dew point within 5 K of ambient -> switch to heating
	ELSIF in_Cryo_Stat.lrDewPointTempC >= (in_Cryo_Stat.lrAmbiantTempC - 5.0) THEN
		nNextState := E_MET_CRYO_ANTI_FOGGING_STATE.HEATING;

	// 4. Dew point within 10 K of ambient -> switch to air blowing
	ELSIF in_Cryo_Stat.lrDewPointTempC >= (in_Cryo_Stat.lrAmbiantTempC - 10.0) THEN
		nNextState := E_MET_CRYO_ANTI_FOGGING_STATE.AIR_BLOWING;

	// 5. All good -> continue standard mode
	ELSE
		nNextState := E_MET_CRYO_ANTI_FOGGING_STATE.STANDARD_OPERATION;
	END_IF

ELSE
	// Manual interrupt
	nNextState := E_MET_CRYO_ANTI_FOGGING_STATE.FINISHED;
END_IF

// Conditional logging: only log if state changes
IF nNextState <> prevState THEN
	CASE nNextState OF
		E_MET_CRYO_ANTI_FOGGING_STATE.ALARM_CONDITION:
			logs.M_LogWarning('Anti-Fogging alarm condition: Dew point dangerously close to window temperature.');
			stat.sState := 'Alarm condition: Dew point close to window temperature.';
		E_MET_CRYO_ANTI_FOGGING_STATE.HEATING:
			logs.M_LogInfo('Anti-Fogging: Starting active heating above dew point.');
			stat.sState := 'Active heating above dew point....';
		E_MET_CRYO_ANTI_FOGGING_STATE.AIR_BLOWING:
			logs.M_LogInfo('Anti-Fogging: Starting air blower (dew point < 10 K below ambient).');
			stat.sState := 'Blowing Air (dew point < 10 K below ambient)...';
		E_MET_CRYO_ANTI_FOGGING_STATE.STANDARD_OPERATION:
			logs.M_LogInfo('Anti-Fogging: Starting standard operation mode.');
			stat.sState := 'Standard operation mode...';
		E_MET_CRYO_ANTI_FOGGING_STATE.FINISHED:
			logs.M_LogInfo('Anti-Fogging routine finished (cryostat warm or operator interrupt).');
	END_CASE
END_IF
END_METHOD

METHOD M_ExecuteControllers
VAR_INPUT
END_VAR
// note: we do not write the auto-enable input (in_bEnable),
// because we call the M_SetEnable and M_SetDisable methods instead
dryair_blow_valve(in_sName:= 'AntiFog Blower Valve', 
				in_eValveType:= E_METIS_CRYO_CTRL_VALVE_TYPE.ANTI_FOG_BLOWER, 
				in_sAutoSetpointSource:= 'Simulated set point');
END_METHOD

METHOD M_HandleEvents
VAR_INPUT
END_VAR

//
// Handle triggers
//

trigEnable	(CLK := ctrl.bEnable);
trigDisable	(CLK := ctrl.bEnable);
END_METHOD

METHOD PRIVATE M_SetError
VAR_INPUT
    nCode     : UDINT;
    sMessage  : STRING;
END_VAR


stat.Error.nCode := nCode;
stat.Error.sMessage := sMessage;
stat.bError := TRUE;
stat.nState := E_MET_CRYO_ANTI_FOGGING_STATE.ERROR;
END_METHOD

METHOD M_Start_AntiFogging : BOOL
VAR_INPUT
END_VAR
ctrl.bEnable := TRUE;
END_METHOD

METHOD M_StateMachine
VAR_INPUT
END_VAR
VAR_IN_OUT
	{attribute 'OPC.UA.DA' := '0'}
	all_cryo_temps:					FB_METIS_TEMPERATURES;
	{attribute 'OPC.UA.DA' := '0'}
	all_heaters:					FB_METIS_HEATERS;
	{attribute 'OPC.UA.DA' := '0'}
	all_t_ctrls:      				FB_METIS_TCTRL;
	{attribute 'OPC.UA.DA' := '0'}
	all_t_votes: 					FB_METIS_VOTERS;
	{attribute 'OPC.UA.DA' := '0'}
	interlocks:						T_METIS_CRYO_INTERLOCKS;
END_VAR


//--- State Machine Logic ---
CASE stat.nState OF
	
	E_MET_CRYO_ANTI_FOGGING_STATE.NONE:
	
		M_Activity_None(		
						all_cryo_temps:= all_cryo_temps,
						all_heaters := all_heaters,
						all_t_ctrls := all_t_ctrls,
						all_t_votes := all_t_votes,
						interlocks := interlocks);
		
	E_MET_CRYO_ANTI_FOGGING_STATE.CHECK_PRECONDITIONS:
	
		M_Activity_Check_Preconditions(		
						all_cryo_temps:= all_cryo_temps,
						all_heaters := all_heaters,
						all_t_ctrls := all_t_ctrls,
						all_t_votes := all_t_votes,
						interlocks := interlocks);
		
	E_MET_CRYO_ANTI_FOGGING_STATE.START_ANTI_FOGGING:
 
		M_Activity_Start_Anti_Fogging(		
						all_cryo_temps:= all_cryo_temps,
						all_heaters := all_heaters,
						all_t_ctrls := all_t_ctrls,
						all_t_votes := all_t_votes,
						interlocks := interlocks);

	E_MET_CRYO_ANTI_FOGGING_STATE.STANDARD_OPERATION:
	
		M_Activity_Standard_Operation(		
						all_cryo_temps:= all_cryo_temps,
						all_heaters := all_heaters,
						all_t_ctrls := all_t_ctrls,
						all_t_votes := all_t_votes,
						interlocks := interlocks);
	
	E_MET_CRYO_ANTI_FOGGING_STATE.AIR_BLOWING:
 
		M_Activity_AirBlowing(		
						all_cryo_temps:= all_cryo_temps,
						all_heaters := all_heaters,
						all_t_ctrls := all_t_ctrls,
						all_t_votes := all_t_votes,
						interlocks := interlocks);

	E_MET_CRYO_ANTI_FOGGING_STATE.HEATING:
	
		M_Activity_Heating(		
						all_cryo_temps:= all_cryo_temps,
						all_heaters := all_heaters,
						all_t_ctrls := all_t_ctrls,
						all_t_votes := all_t_votes,
						interlocks := interlocks);
						
	E_MET_CRYO_ANTI_FOGGING_STATE.ALARM_CONDITION: 
		M_Activity_Alarm_Condition(		
						all_cryo_temps:= all_cryo_temps,
						all_heaters := all_heaters,
						all_t_ctrls := all_t_ctrls,
						all_t_votes := all_t_votes,
						interlocks := interlocks);
	E_MET_CRYO_ANTI_FOGGING_STATE.FINISHED: 
	
		M_Activity_Finished(		
						all_cryo_temps:= all_cryo_temps,
						all_heaters := all_heaters,
						all_t_ctrls := all_t_ctrls,
						all_t_votes := all_t_votes,
						interlocks := interlocks);
	
	E_MET_CRYO_ANTI_FOGGING_STATE.ERROR:
		
		M_Activity_Error_Handling(		
						all_cryo_temps:= all_cryo_temps,
						all_heaters := all_heaters,
						all_t_ctrls := all_t_ctrls,
						all_t_votes := all_t_votes,
						interlocks := interlocks);
		
END_CASE;
END_METHOD

METHOD M_Stop_AntiFogging : BOOL
VAR_INPUT
END_VAR
ctrl.bEnable := FALSE;
END_METHOD

METHOD M_UpdateStatus
VAR_INPUT
END_VAR
VAR_IN_OUT
	{attribute 'OPC.UA.DA' := '0'}
	all_cryo_temps:					FB_METIS_TEMPERATURES;
	{attribute 'OPC.UA.DA' := '0'}
	all_heaters:					FB_METIS_HEATERS;
	{attribute 'OPC.UA.DA' := '0'}
	all_t_ctrls:      				FB_METIS_TCTRL;
	{attribute 'OPC.UA.DA' := '0'}
	all_t_votes: 					FB_METIS_VOTERS;
	{attribute 'OPC.UA.DA' := '0'}
	interlocks:						T_METIS_CRYO_INTERLOCKS;
END_VAR


IF stat.nState = E_MET_CRYO_ANTI_FOGGING_STATE.ERROR THEN
	stat.bError := TRUE;
ELSE
	stat.bError := FALSE;
END_IF



out_bAntiFoggingActive := stat.bActive;
stat.bBusy := stat.bActive;


 //Check Pre-Conditions for HMI Enable 
stat.bPreConditionsMet := 	(in_Cryo_Stat.bInVacuum OR in_Cryo_Stat.bInGoodVacuum) AND
							(NOT in_Cryo_Stat.bWarm);
END_METHOD

END_FUNCTION_BLOCK

// POUs/Devices/Temperature/FB_METIS_TEMPERATURES
FUNCTION_BLOCK FB_METIS_TEMPERATURES
VAR_OUTPUT
	out_lrHighestTemp:		LREAL;
	out_sHighestTempName:	STRING;
	out_bHighestTempValid:	BOOL;
	
	out_lrLowestTemp:		LREAL;
	out_sLowestTempName:	STRING;
	out_bLowestTempValid:	BOOL;
	
	out_lrAverageOfAllTemps: LREAL;
	
	out_all_temperature_names   : ARRAY [0..134] OF STRING;
END_VAR
VAR
	
	{attribute 'OPC.UA.DA' := '0'}
	{attribute 'TcHmiSymbol.Show'}
	all_temperatures		: ARRAY [MIN_INDEX..MAX_INDEX] OF POINTER TO FB_METIS_TEMPERATURE;
    
    // NOTE: the names below are needed for the VISU, which cannot deal with MIN_INDEX and MAX_INDEX
    // Hence, we must specify the numbers explicitly
    // MAKE SURE THE INDEXES ALWATS CORRESPOND TO THE CONSTANTS MIN_INDEX AND MAX_INDEX
	{attribute 'OPC.UA.DA' := '0'}
	{attribute 'TcHmiSymbol.Show'}
    all_temperature_names   : ARRAY [0..134] OF STRING;  // names of the temperatures

(* Empty temp: 1 *)
    
{attribute 'OPC.UA.DA' := '0'}
empty_temp					: FB_METIS_TEMPERATURE;

(*Temp Cryo: 23 + 10 = 33 *)
{attribute 'TcHmiSymbol.Show'}
t_cry_sha_1 				:FB_METIS_TEMPERATURE;
{attribute 'TcHmiSymbol.Show'}
t_cry_sha_2					:FB_METIS_TEMPERATURE;
{attribute 'TcHmiSymbol.Show'}
t_cry_sha_3					:FB_METIS_TEMPERATURE;
{attribute 'TcHmiSymbol.Show'}
t_cry_sha_4                	:FB_METIS_TEMPERATURE;
{attribute 'TcHmiSymbol.Show'}
t_cry_shb_1					:FB_METIS_TEMPERATURE;
{attribute 'TcHmiSymbol.Show'}
t_cry_shb_2                	:FB_METIS_TEMPERATURE;
t_cry_shb_3                	:FB_METIS_TEMPERATURE;
t_cry_shb_4                	:FB_METIS_TEMPERATURE;
t_cry_shc_1					:FB_METIS_TEMPERATURE;
t_cry_shc_2                	:FB_METIS_TEMPERATURE;
t_cry_shc_3                	:FB_METIS_TEMPERATURE;
t_cry_shc_4                	:FB_METIS_TEMPERATURE;
t_cry_pta_1                	:FB_METIS_TEMPERATURE;
t_cry_pta_2                	:FB_METIS_TEMPERATURE;
t_cry_ptb_1                	:FB_METIS_TEMPERATURE;
t_cry_ptb_2                	:FB_METIS_TEMPERATURE;
t_cry_ptc_1					:FB_METIS_TEMPERATURE;
t_cry_ptc_2                	:FB_METIS_TEMPERATURE;
t_cry_pta_3                	:FB_METIS_TEMPERATURE;
t_cry_ptb_3                	:FB_METIS_TEMPERATURE;
t_cry_ptc_3                	:FB_METIS_TEMPERATURE;
{attribute 'TcHmiSymbol.Show'}
t_cry_sp_1					:FB_METIS_TEMPERATURE;
{attribute 'TcHmiSymbol.Show'}
t_cry_sp_2					:FB_METIS_TEMPERATURE;
// voter outputs 
t_cry_vot_1                 :FB_METIS_TEMPERATURE;
t_cry_vot_2                 :FB_METIS_TEMPERATURE;
t_cry_vot_3                 :FB_METIS_TEMPERATURE;
t_cry_vot_4                 :FB_METIS_TEMPERATURE;
t_cry_vot_5                 :FB_METIS_TEMPERATURE;
t_cry_vot_6                 :FB_METIS_TEMPERATURE;
t_cry_vot_7                 :FB_METIS_TEMPERATURE;
t_cry_vot_8                 :FB_METIS_TEMPERATURE;
t_cry_vot_9                 :FB_METIS_TEMPERATURE;
t_cry_vot_10                :FB_METIS_TEMPERATURE;
                            
(*SCA Temps: 16 + 4 + 10 + 3 = 33 *)  
         
// cu X2
t_sca_fw_1                  :FB_METIS_TEMPERATURE;
t_sca_fw_2                  :FB_METIS_TEMPERATURE;
t_sca_lu_1                  :FB_METIS_TEMPERATURE;
t_sca_fm                    :FB_METIS_TEMPERATURE;
t_sca_fs                    :FB_METIS_TEMPERATURE;
t_sca_lu_2                  :FB_METIS_TEMPERATURE;
t_sca_mod                   :FB_METIS_TEMPERATURE;
t_sca_pyr					:FB_METIS_TEMPERATURE;
// cu X3
t_sca_h_1                   :FB_METIS_TEMPERATURE;
t_sca_if_1                  :FB_METIS_TEMPERATURE;
t_sca_if_2                  :FB_METIS_TEMPERATURE;
t_sca_lu_3                  :FB_METIS_TEMPERATURE;
t_sca_bp_1                  :FB_METIS_TEMPERATURE;
t_sca_bp_2                  :FB_METIS_TEMPERATURE;
t_sca_bp_3                  :FB_METIS_TEMPERATURE;
t_sca_h_2                   :FB_METIS_TEMPERATURE;
// detector (4)
t_sca_det_1                 :FB_METIS_TEMPERATURE;
t_sca_det_2                 :FB_METIS_TEMPERATURE;
t_sca_dhs_1                 :FB_METIS_TEMPERATURE;
t_sca_dhs_2                 :FB_METIS_TEMPERATURE;
// voter outputs (10)
t_sca_vot_1                 :FB_METIS_TEMPERATURE;
t_sca_vot_2                 :FB_METIS_TEMPERATURE;
t_sca_vot_3                 :FB_METIS_TEMPERATURE;
t_sca_vot_4                 :FB_METIS_TEMPERATURE;
t_sca_vot_5                 :FB_METIS_TEMPERATURE;
t_sca_vot_6                 :FB_METIS_TEMPERATURE;
t_sca_vot_7                 :FB_METIS_TEMPERATURE;
t_sca_vot_8                 :FB_METIS_TEMPERATURE;
t_sca_vot_9                 :FB_METIS_TEMPERATURE;
t_sca_vot_10                :FB_METIS_TEMPERATURE;
// temperature controller ramps (3)
t_sca_wuh_ramp              :FB_METIS_TEMPERATURE;
t_sca_det_2_ramp            :FB_METIS_TEMPERATURE;
t_sca_dhs_2_ramp            :FB_METIS_TEMPERATURE;




(*IMG Temps : 24 + 6 + 10 + 4 = 44 *)              

// cu (24)
t_img_lpw_1                 :FB_METIS_TEMPERATURE;
t_img_lpw_2                 :FB_METIS_TEMPERATURE;
t_img_lfw_1                 :FB_METIS_TEMPERATURE;
t_img_lfw_2                 :FB_METIS_TEMPERATURE;
t_img_lpr_1                 :FB_METIS_TEMPERATURE;
t_img_bwu_3                 :FB_METIS_TEMPERATURE;
t_img_lnd_1                 :FB_METIS_TEMPERATURE;
t_img_lnd_2                 :FB_METIS_TEMPERATURE;
t_img_npw_1                 :FB_METIS_TEMPERATURE;
t_img_npw_2                 :FB_METIS_TEMPERATURE;
t_img_nfw_1                 :FB_METIS_TEMPERATURE;
t_img_nfw_2                 :FB_METIS_TEMPERATURE;
t_img_npr_1                 :FB_METIS_TEMPERATURE;
t_img_bwu_2                 :FB_METIS_TEMPERATURE;
t_img_nnd_1                 :FB_METIS_TEMPERATURE;
t_img_nnd_2                 :FB_METIS_TEMPERATURE;
t_img_opt_1                 :FB_METIS_TEMPERATURE;
t_img_bwu_1                 :FB_METIS_TEMPERATURE;
t_img_ctr_1                 :FB_METIS_TEMPERATURE;
t_img_ctr_2                 :FB_METIS_TEMPERATURE;
t_img_70k_1                 :FB_METIS_TEMPERATURE;
t_img_ln2_1                 :FB_METIS_TEMPERATURE;
t_img_ln2_2				    :FB_METIS_TEMPERATURE;
t_img_hex_1                 :FB_METIS_TEMPERATURE;
// detector (6)
t_img_lmd_1                 :FB_METIS_TEMPERATURE;
t_img_lmd_2                 :FB_METIS_TEMPERATURE;
t_img_lmp_1                 :FB_METIS_TEMPERATURE;
t_img_lmp_2                 :FB_METIS_TEMPERATURE;
t_img_nd_1                  :FB_METIS_TEMPERATURE;
t_img_nd_2                  :FB_METIS_TEMPERATURE;
// voter outputs (10)
t_img_vot_1                 :FB_METIS_TEMPERATURE;
t_img_vot_2                 :FB_METIS_TEMPERATURE;
t_img_vot_3                 :FB_METIS_TEMPERATURE;
t_img_vot_4                 :FB_METIS_TEMPERATURE;
t_img_vot_5                 :FB_METIS_TEMPERATURE;
t_img_vot_6                 :FB_METIS_TEMPERATURE;
t_img_vot_7                 :FB_METIS_TEMPERATURE;
t_img_vot_8                 :FB_METIS_TEMPERATURE;
t_img_vot_9                 :FB_METIS_TEMPERATURE;
t_img_vot_10                :FB_METIS_TEMPERATURE;
// temperature controller ramps (4)
t_img_wuh_ramp              :FB_METIS_TEMPERATURE;
t_img_lmd_2_ramp            :FB_METIS_TEMPERATURE;
t_img_lmp_2_ramp            :FB_METIS_TEMPERATURE;
t_img_nd_2_ramp             :FB_METIS_TEMPERATURE;
                            
(*Temp LMS : 16 *)  
                            
t_lms_pma_1                 :FB_METIS_TEMPERATURE;
t_lms_pma_2                 :FB_METIS_TEMPERATURE;
t_lms_msa_1                 :FB_METIS_TEMPERATURE;
t_lms_msa_2                 :FB_METIS_TEMPERATURE;
t_lms_pra_1                 :FB_METIS_TEMPERATURE;
t_lms_pra_2                 :FB_METIS_TEMPERATURE;
t_lms_gra_1                 :FB_METIS_TEMPERATURE;
t_lms_gra_2                 :FB_METIS_TEMPERATURE;
t_lms_pla_1                 :FB_METIS_TEMPERATURE;
t_lms_pla_2                 :FB_METIS_TEMPERATURE;
t_lms_pla_3                 :FB_METIS_TEMPERATURE;
t_lms_pla_4                 :FB_METIS_TEMPERATURE;
t_lms_tma                   :FB_METIS_TEMPERATURE;
t_lms_dtw                   :FB_METIS_TEMPERATURE;
t_lms_ptw                   :FB_METIS_TEMPERATURE;
t_lms_spare                 :FB_METIS_TEMPERATURE;
                            
(*Temp CFO*) 


// RTD temperatures
t_cry_pca                   : FB_METIS_TEMPERATURE; // PCA.T = IMG Heat Exchanger Out
t_cry_pcb                   : FB_METIS_TEMPERATURE; // PCB.T = CFO Heat Exchanger Out
t_cry_wim                   : FB_METIS_TEMPERATURE; // WI.MT = Window Mount
t_cry_wia                   : FB_METIS_TEMPERATURE; // WI.AT = Window Ambient
// dew point temperatures
t_cry_wid                   : FB_METIS_TEMPERATURE;

(*System temperatures   (3) *)
// Master temperature to estimate overall temperature of the cryostat  
t_master                 	:FB_METIS_TEMPERATURE;
t_master_vot_1           	:FB_METIS_TEMPERATURE;
t_master_vot_2           	:FB_METIS_TEMPERATURE;


(*Vars*)

{attribute 'OPC.UA.DA' := '0'}
bConfigured					: BOOL := FALSE;

(*Temperature Simulation*)

sim_t_cry_sha_1: 		FB_SIM_TEMP_SENSOR_DT670;
sim_t_cry_sha_2: 		FB_SIM_TEMP_SENSOR_DT670; 
sim_t_sca_fw_icar: 		FB_SIM_TEMP_SENSOR_DT670;
sim_t_img_n_pw_icar: 	FB_SIM_TEMP_SENSOR_DT670;
sim_t_lms_pla_1: 		FB_SIM_TEMP_SENSOR_DT670;
               
END_VAR
VAR CONSTANT
	{attribute 'OPC.UA.DA' := '0'}
    MIN_INDEX : INT := 0;
	{attribute 'OPC.UA.DA' := '0'}
    MAX_INDEX : INT := 134; // 1 + 33 + 33 + 44 + 16 + 5 + 3 = 135 items ==> MAX_INDEX = 134
END_VAR

M_Configure();

// to avoid invalid pointers, it is recommended to update the pointers every cycle
M_UpdatePointers();

M_ReadSensors();

M_MaxMinAvrgTemperatures();


//sim_t_cry_sha_1(in_Temp_Sensor_DT670 := t_cry_sha_1);
//sim_t_cry_sha_2(in_Temp_Sensor_DT670 := t_cry_sha_2);
//sim_t_sca_fw_icar(in_Temp_Sensor_DT670 := t_sca_fw_icar);
//sim_t_img_n_pw_icar(in_Temp_Sensor_DT670 := t_img_n_pw_icar);
//sim_t_lms_pla_1(in_Temp_Sensor_DT670 := t_lms_pla_1);

METHOD M_ConfigSimTemperatures
VAR_INPUT
END_VAR


//sim_t_cry_sha_1(in_Temp_Sensor_DT670 := t_cry_sha_1);
//sim_t_cry_sha_2(in_Temp_Sensor_DT670 := t_cry_sha_2);
//sim_t_sca_fw_icar(in_Temp_Sensor_DT670 := t_sca_fw_icar);
//sim_t_img_n_pw_icar(in_Temp_Sensor_DT670 := t_img_n_pw_icar);
//sim_t_lms_pla_1(in_Temp_Sensor_DT670 := t_lms_pla_1);
END_METHOD

METHOD M_Configure : BOOL
VAR_INPUT
END_VAR
VAR
    i : INT;
END_VAR
IF NOT bConfigured THEN
    
    // just as a safety precaution, set valid pointers to start with
    FOR i := MIN_INDEX TO MAX_INDEX DO
        all_temperatures[i] := ADR(empty_temp);
    END_FOR
    
    // Configure the all temp array
    M_UpdatePointers();
    
    // execute the M_ReadSensors function once to update the names
    M_ReadSensors();
    
    // store the names in a separate array
    FOR i := MIN_INDEX TO MAX_INDEX DO
        all_temperature_names[i] := all_temperatures[i]^.in_sName;
    END_FOR

    // Config SIM Temperatures
    M_ConfigSimTemperatures();
    
    bConfigured := TRUE;
END_IF
END_METHOD

METHOD M_GetTempSensorIndex : INT
VAR_INPUT
    sName : STRING;
END_VAR
VAR
    i: INT;
END_VAR
FOR i := MIN_INDEX TO MAX_INDEX DO
    IF sName = all_temperatures[i]^.in_sName THEN
        M_GetTempSensorIndex := i;
        RETURN;
    END_IF
END_FOR

// Handle error: sensor name not found
M_GetTempSensorIndex := 0; // empty temperature
END_METHOD

METHOD M_IsIgnoredTemperature : BOOL
VAR_INPUT
    index : INT;   // Index into all_temperatures[]
END_VAR
VAR

    IgnoreList: 		ARRAY[1..5] OF STRING := [
        't_cry_pca',
        't_cry_pcb',
        't_cry_wim',
        't_cry_wia',
        't_cry_wid'
    ];
    i : INT;
END_VAR
M_IsIgnoredTemperature := FALSE;

// Loop through ignore list
FOR i := 1 TO 5 DO
    IF all_temperatures[index]^.in_sName = IgnoreList[i] THEN
        M_IsIgnoredTemperature := TRUE;
        RETURN; // Exit early once a match is found
    END_IF
END_FOR
END_METHOD

METHOD M_MaxMinAvrgTemperatures
VAR_INPUT
END_VAR
VAR
	lrHigestTemp:		LREAL;	// Temporary var Higest temp
	sHighestTempName:	STRING;
	
	lrLowestTemp:		LREAL;	// Temporary var Lowest temp
	sLowestTempName:	STRING;
	
	lrAverageTemp:		LREAL;	// Temporary var Lowest temp
	nSample:	INT;	// Number of valid sensor readings
	i:			INT;
	
	
END_VAR
(*Highest Temperature*)

lrHigestTemp	:= -10000.0; // setting initial temperature for comparision
sHighestTempName := '';
lrLowestTemp := 10000.0; // setting initial temperature for comparision
sLowestTempName := '';
lrAverageTemp:= 0.0; 	// setting initial temperature for comparision		

nSample	:= 0;

FOR i := MIN_INDEX TO MAX_INDEX DO
		// Ignor Ambient temps
		IF M_IsIgnoredTemperature(index := i) THEN		
			; // Skip this sensor in averaging, highest, lowest calculation
		ELSE			
			IF  all_temperatures[i]^.stat.bValid	THEN
				
					IF  all_temperatures[i]^.stat.lrTempK > lrHigestTemp THEN
						lrHigestTemp	:= all_temperatures[i]^.stat.lrTempK;
						sHighestTempName := all_temperatures[i]^.in_sName;
					END_IF
					
					IF  all_temperatures[i]^.stat.lrTempK < lrLowestTemp THEN
						lrLowestTemp	:= all_temperatures[i]^.stat.lrTempK;
						sLowestTempName    := all_temperatures[i]^.in_sName;
					END_IF
					
					lrAverageTemp	:= lrAverageTemp + all_temperatures[i]^.stat.lrTempK;	
					
					nSample	:= nSample + 1;
			END_IF
			
		END_IF
END_FOR



IF nSample > 0	THEN
	out_lrAverageOfAllTemps	:= lrAverageTemp / nSample;
	
	out_lrHighestTemp := lrHigestTemp;		
	out_sHighestTempName := sHighestTempName;
	out_bHighestTempValid := TRUE;
	
	out_lrLowestTemp :=		lrLowestTemp;
	out_sLowestTempName :=	sLowestTempName;
	out_bLowestTempValid := TRUE;
	
	
	
ELSE
	
	out_lrAverageOfAllTemps	:= 9999;
	
	out_lrHighestTemp := 9999;		
	out_sHighestTempName := 'NA';
	out_bHighestTempValid := FALSE;
	
	out_lrLowestTemp :=		9999;
	out_sLowestTempName :=	'NA';
	out_bLowestTempValid := FALSE;
END_IF
END_METHOD

METHOD M_ReadSensors
VAR_INPUT
END_VAR
empty_temp			(in_sName:='', in_eType := E_METIS_SENSOR_TYPE.TEMPERATURE, in_eSource := E_METIS_SENSOR_SOURCE.LS240, in_nRampPeriodSec:= 10, in_lrFaultRamp:= 10);
	

t_cry_sha_1			(in_sName:='t_cry_sha_1', in_eType := E_METIS_SENSOR_TYPE.TEMPERATURE, in_eSource := E_METIS_SENSOR_SOURCE.LS240, in_nRampPeriodSec:= 10, in_lrFaultRamp:= 10);
t_cry_sha_2			(in_sName:='t_cry_sha_2', in_eType := E_METIS_SENSOR_TYPE.TEMPERATURE, in_eSource := E_METIS_SENSOR_SOURCE.LS240, in_nRampPeriodSec:= 10, in_lrFaultRamp:= 10);			
t_cry_sha_3			(in_sName:='t_cry_sha_3', in_eType := E_METIS_SENSOR_TYPE.TEMPERATURE, in_eSource := E_METIS_SENSOR_SOURCE.LS240, in_nRampPeriodSec:= 10, in_lrFaultRamp:= 10);	
t_cry_sha_4		    (in_sName:='t_cry_sha_4', in_eType := E_METIS_SENSOR_TYPE.TEMPERATURE, in_eSource := E_METIS_SENSOR_SOURCE.LS240, in_nRampPeriodSec:= 10, in_lrFaultRamp:= 10);    
t_cry_shb_1			(in_sName:='t_cry_shb_1', in_eType := E_METIS_SENSOR_TYPE.TEMPERATURE, in_eSource := E_METIS_SENSOR_SOURCE.LS240, in_nRampPeriodSec:= 10, in_lrFaultRamp:= 10);	
t_cry_shb_2		    (in_sName:='t_cry_shb_2', in_eType := E_METIS_SENSOR_TYPE.TEMPERATURE, in_eSource := E_METIS_SENSOR_SOURCE.LS240, in_nRampPeriodSec:= 10, in_lrFaultRamp:= 10);    
t_cry_shb_3		    (in_sName:='t_cry_shb_3', in_eType := E_METIS_SENSOR_TYPE.TEMPERATURE, in_eSource := E_METIS_SENSOR_SOURCE.LS240, in_nRampPeriodSec:= 10, in_lrFaultRamp:= 10);   
t_cry_shb_4			(in_sName:='t_cry_shb_4', in_eType := E_METIS_SENSOR_TYPE.TEMPERATURE, in_eSource := E_METIS_SENSOR_SOURCE.LS240, in_nRampPeriodSec:= 10, in_lrFaultRamp:= 10);            
t_cry_shc_1			(in_sName:='t_cry_shc_1', in_eType := E_METIS_SENSOR_TYPE.TEMPERATURE, in_eSource := E_METIS_SENSOR_SOURCE.LS240, in_nRampPeriodSec:= 10, in_lrFaultRamp:= 10);	
t_cry_shc_2		    (in_sName:='t_cry_shc_2', in_eType := E_METIS_SENSOR_TYPE.TEMPERATURE, in_eSource := E_METIS_SENSOR_SOURCE.LS240, in_nRampPeriodSec:= 10, in_lrFaultRamp:= 10);    
t_cry_shc_3		    (in_sName:='t_cry_shc_3', in_eType := E_METIS_SENSOR_TYPE.TEMPERATURE, in_eSource := E_METIS_SENSOR_SOURCE.LS240, in_nRampPeriodSec:= 10, in_lrFaultRamp:= 10);    
t_cry_shc_4		    (in_sName:='t_cry_shc_4', in_eType := E_METIS_SENSOR_TYPE.TEMPERATURE, in_eSource := E_METIS_SENSOR_SOURCE.LS240, in_nRampPeriodSec:= 10, in_lrFaultRamp:= 10);    
t_cry_pta_1		    (in_sName:='t_cry_pta_1', in_eType := E_METIS_SENSOR_TYPE.TEMPERATURE, in_eSource := E_METIS_SENSOR_SOURCE.LS240, in_nRampPeriodSec:= 10, in_lrFaultRamp:= 10);    
t_cry_pta_2		    (in_sName:='t_cry_pta_2', in_eType := E_METIS_SENSOR_TYPE.TEMPERATURE, in_eSource := E_METIS_SENSOR_SOURCE.LS240, in_nRampPeriodSec:= 10, in_lrFaultRamp:= 10);    
t_cry_ptb_1		    (in_sName:='t_cry_ptb_1', in_eType := E_METIS_SENSOR_TYPE.TEMPERATURE, in_eSource := E_METIS_SENSOR_SOURCE.LS240, in_nRampPeriodSec:= 10, in_lrFaultRamp:= 10);    
t_cry_ptb_2		    (in_sName:='t_cry_ptb_2', in_eType := E_METIS_SENSOR_TYPE.TEMPERATURE, in_eSource := E_METIS_SENSOR_SOURCE.LS240, in_nRampPeriodSec:= 10, in_lrFaultRamp:= 10);    
t_cry_ptc_1			(in_sName:='t_cry_ptc_1', in_eType := E_METIS_SENSOR_TYPE.TEMPERATURE, in_eSource := E_METIS_SENSOR_SOURCE.LS240, in_nRampPeriodSec:= 10, in_lrFaultRamp:= 10);	
t_cry_ptc_2		    (in_sName:='t_cry_ptc_2', in_eType := E_METIS_SENSOR_TYPE.TEMPERATURE, in_eSource := E_METIS_SENSOR_SOURCE.LS240, in_nRampPeriodSec:= 10, in_lrFaultRamp:= 10);    
t_cry_pta_3		    (in_sName:='t_cry_pta_3', in_eType := E_METIS_SENSOR_TYPE.TEMPERATURE, in_eSource := E_METIS_SENSOR_SOURCE.LS240, in_nRampPeriodSec:= 10, in_lrFaultRamp:= 10);    
t_cry_ptb_3		    (in_sName:='t_cry_ptb_3', in_eType := E_METIS_SENSOR_TYPE.TEMPERATURE, in_eSource := E_METIS_SENSOR_SOURCE.LS240, in_nRampPeriodSec:= 10, in_lrFaultRamp:= 10);    
t_cry_ptc_3		    (in_sName:='t_cry_ptc_3', in_eType := E_METIS_SENSOR_TYPE.TEMPERATURE, in_eSource := E_METIS_SENSOR_SOURCE.LS240, in_nRampPeriodSec:= 10, in_lrFaultRamp:= 10);    
t_cry_sp_1			(in_sName:='t_cry_sp_1',  in_eType := E_METIS_SENSOR_TYPE.TEMPERATURE, in_eSource := E_METIS_SENSOR_SOURCE.LS240, in_nRampPeriodSec:= 10, in_lrFaultRamp:= 10);
t_cry_sp_2			(in_sName:='t_cry_sp_2',  in_eType := E_METIS_SENSOR_TYPE.TEMPERATURE, in_eSource := E_METIS_SENSOR_SOURCE.LS240, in_nRampPeriodSec:= 10, in_lrFaultRamp:= 10);
t_cry_vot_1         (in_sName:='t_cry_vot_1',  in_eType := E_METIS_SENSOR_TYPE.TEMPERATURE, in_eSource := E_METIS_SENSOR_SOURCE.VOTER, in_nRampPeriodSec:= 10, in_lrFaultRamp:= 10);
t_cry_vot_2         (in_sName:='t_cry_vot_2',  in_eType := E_METIS_SENSOR_TYPE.TEMPERATURE, in_eSource := E_METIS_SENSOR_SOURCE.VOTER, in_nRampPeriodSec:= 10, in_lrFaultRamp:= 10);
t_cry_vot_3         (in_sName:='t_cry_vot_3',  in_eType := E_METIS_SENSOR_TYPE.TEMPERATURE, in_eSource := E_METIS_SENSOR_SOURCE.VOTER, in_nRampPeriodSec:= 10, in_lrFaultRamp:= 10);
t_cry_vot_4         (in_sName:='t_cry_vot_4',  in_eType := E_METIS_SENSOR_TYPE.TEMPERATURE, in_eSource := E_METIS_SENSOR_SOURCE.VOTER, in_nRampPeriodSec:= 10, in_lrFaultRamp:= 10);
t_cry_vot_5         (in_sName:='t_cry_vot_5',  in_eType := E_METIS_SENSOR_TYPE.TEMPERATURE, in_eSource := E_METIS_SENSOR_SOURCE.VOTER, in_nRampPeriodSec:= 10, in_lrFaultRamp:= 10);
t_cry_vot_6         (in_sName:='t_cry_vot_6',  in_eType := E_METIS_SENSOR_TYPE.TEMPERATURE, in_eSource := E_METIS_SENSOR_SOURCE.VOTER, in_nRampPeriodSec:= 10, in_lrFaultRamp:= 10);
t_cry_vot_7         (in_sName:='t_cry_vot_7',  in_eType := E_METIS_SENSOR_TYPE.TEMPERATURE, in_eSource := E_METIS_SENSOR_SOURCE.VOTER, in_nRampPeriodSec:= 10, in_lrFaultRamp:= 10);
t_cry_vot_8         (in_sName:='t_cry_vot_8',  in_eType := E_METIS_SENSOR_TYPE.TEMPERATURE, in_eSource := E_METIS_SENSOR_SOURCE.VOTER, in_nRampPeriodSec:= 10, in_lrFaultRamp:= 10);
t_cry_vot_9         (in_sName:='t_cry_vot_9',  in_eType := E_METIS_SENSOR_TYPE.TEMPERATURE, in_eSource := E_METIS_SENSOR_SOURCE.VOTER, in_nRampPeriodSec:= 10, in_lrFaultRamp:= 10);
t_cry_vot_10        (in_sName:='t_cry_vot_10', in_eType := E_METIS_SENSOR_TYPE.TEMPERATURE, in_eSource := E_METIS_SENSOR_SOURCE.VOTER, in_nRampPeriodSec:= 10, in_lrFaultRamp:= 10);                       

	(*SCA Temps*)   
	
t_sca_fw_1          (in_sName:='t_sca_fw_1',    in_eType := E_METIS_SENSOR_TYPE.TEMPERATURE, in_eSource := E_METIS_SENSOR_SOURCE.LS240, in_nRampPeriodSec:= 10, in_lrFaultRamp:= 10);    
t_sca_fw_2          (in_sName:='t_sca_fw_2',    in_eType := E_METIS_SENSOR_TYPE.TEMPERATURE, in_eSource := E_METIS_SENSOR_SOURCE.LS240, in_nRampPeriodSec:= 10, in_lrFaultRamp:= 10);    
t_sca_lu_1          (in_sName:='t_sca_lu_1',    in_eType := E_METIS_SENSOR_TYPE.TEMPERATURE, in_eSource := E_METIS_SENSOR_SOURCE.LS240, in_nRampPeriodSec:= 10, in_lrFaultRamp:= 10);    
t_sca_fm            (in_sName:='t_sca_fm', 	    in_eType := E_METIS_SENSOR_TYPE.TEMPERATURE, in_eSource := E_METIS_SENSOR_SOURCE.LS240, in_nRampPeriodSec:= 10, in_lrFaultRamp:= 10);    
t_sca_fs            (in_sName:='t_sca_fs',      in_eType := E_METIS_SENSOR_TYPE.TEMPERATURE, in_eSource := E_METIS_SENSOR_SOURCE.LS240, in_nRampPeriodSec:= 10, in_lrFaultRamp:= 10);    
t_sca_lu_2          (in_sName:='t_sca_lu_2',    in_eType := E_METIS_SENSOR_TYPE.TEMPERATURE, in_eSource := E_METIS_SENSOR_SOURCE.LS240, in_nRampPeriodSec:= 10, in_lrFaultRamp:= 10);    
t_sca_mod           (in_sName:='t_sca_mod',     in_eType := E_METIS_SENSOR_TYPE.TEMPERATURE, in_eSource := E_METIS_SENSOR_SOURCE.LS240, in_nRampPeriodSec:= 10, in_lrFaultRamp:= 10);    
t_sca_pyr			(in_sName:='t_sca_pyr',     in_eType := E_METIS_SENSOR_TYPE.TEMPERATURE, in_eSource := E_METIS_SENSOR_SOURCE.LS240, in_nRampPeriodSec:= 10, in_lrFaultRamp:= 10);	
t_sca_h_1           (in_sName:='t_sca_h_1',     in_eType := E_METIS_SENSOR_TYPE.TEMPERATURE, in_eSource := E_METIS_SENSOR_SOURCE.LS240, in_nRampPeriodSec:= 10, in_lrFaultRamp:= 10);    
t_sca_if_1          (in_sName:='t_sca_if_1',    in_eType := E_METIS_SENSOR_TYPE.TEMPERATURE, in_eSource := E_METIS_SENSOR_SOURCE.LS240, in_nRampPeriodSec:= 10, in_lrFaultRamp:= 10);    
t_sca_if_2          (in_sName:='t_sca_if_2',    in_eType := E_METIS_SENSOR_TYPE.TEMPERATURE, in_eSource := E_METIS_SENSOR_SOURCE.LS240, in_nRampPeriodSec:= 10, in_lrFaultRamp:= 10);    
t_sca_lu_3          (in_sName:='t_sca_lu_3',    in_eType := E_METIS_SENSOR_TYPE.TEMPERATURE, in_eSource := E_METIS_SENSOR_SOURCE.LS240, in_nRampPeriodSec:= 10, in_lrFaultRamp:= 10);    
t_sca_bp_1          (in_sName:='t_sca_bp_1',    in_eType := E_METIS_SENSOR_TYPE.TEMPERATURE, in_eSource := E_METIS_SENSOR_SOURCE.LS240, in_nRampPeriodSec:= 10, in_lrFaultRamp:= 10);    
t_sca_bp_2          (in_sName:='t_sca_bp_2',    in_eType := E_METIS_SENSOR_TYPE.TEMPERATURE, in_eSource := E_METIS_SENSOR_SOURCE.LS240, in_nRampPeriodSec:= 10, in_lrFaultRamp:= 10);    
t_sca_bp_3          (in_sName:='t_sca_bp_3',    in_eType := E_METIS_SENSOR_TYPE.TEMPERATURE, in_eSource := E_METIS_SENSOR_SOURCE.LS240, in_nRampPeriodSec:= 10, in_lrFaultRamp:= 10);    
t_sca_h_2           (in_sName:='t_sca_h_2',     in_eType := E_METIS_SENSOR_TYPE.TEMPERATURE, in_eSource := E_METIS_SENSOR_SOURCE.LS240, in_nRampPeriodSec:= 10, in_lrFaultRamp:= 10);    
t_sca_det_1         (in_sName:='t_sca_det_1',  in_eType := E_METIS_SENSOR_TYPE.TEMPERATURE, in_eSource := E_METIS_SENSOR_SOURCE.LS336, in_nRampPeriodSec:= 10, in_lrFaultRamp:= 10);
t_sca_det_2         (in_sName:='t_sca_det_2',  in_eType := E_METIS_SENSOR_TYPE.TEMPERATURE, in_eSource := E_METIS_SENSOR_SOURCE.LS336, in_nRampPeriodSec:= 10, in_lrFaultRamp:= 10);
t_sca_dhs_1         (in_sName:='t_sca_dhs_1',  in_eType := E_METIS_SENSOR_TYPE.TEMPERATURE, in_eSource := E_METIS_SENSOR_SOURCE.LS336, in_nRampPeriodSec:= 10, in_lrFaultRamp:= 10);
t_sca_dhs_2         (in_sName:='t_sca_dhs_2',  in_eType := E_METIS_SENSOR_TYPE.TEMPERATURE, in_eSource := E_METIS_SENSOR_SOURCE.LS336, in_nRampPeriodSec:= 10, in_lrFaultRamp:= 10);;
t_sca_vot_1         (in_sName:='t_sca_vot_1',  in_eType := E_METIS_SENSOR_TYPE.TEMPERATURE, in_eSource := E_METIS_SENSOR_SOURCE.VOTER, in_nRampPeriodSec:= 10, in_lrFaultRamp:= 10);
t_sca_vot_2         (in_sName:='t_sca_vot_2',  in_eType := E_METIS_SENSOR_TYPE.TEMPERATURE, in_eSource := E_METIS_SENSOR_SOURCE.VOTER, in_nRampPeriodSec:= 10, in_lrFaultRamp:= 10);
t_sca_vot_3         (in_sName:='t_sca_vot_3',  in_eType := E_METIS_SENSOR_TYPE.TEMPERATURE, in_eSource := E_METIS_SENSOR_SOURCE.VOTER, in_nRampPeriodSec:= 10, in_lrFaultRamp:= 10);
t_sca_vot_4         (in_sName:='t_sca_vot_4',  in_eType := E_METIS_SENSOR_TYPE.TEMPERATURE, in_eSource := E_METIS_SENSOR_SOURCE.VOTER, in_nRampPeriodSec:= 10, in_lrFaultRamp:= 10);
t_sca_vot_5         (in_sName:='t_sca_vot_5',  in_eType := E_METIS_SENSOR_TYPE.TEMPERATURE, in_eSource := E_METIS_SENSOR_SOURCE.VOTER, in_nRampPeriodSec:= 10, in_lrFaultRamp:= 10);
t_sca_vot_6         (in_sName:='t_sca_vot_6',  in_eType := E_METIS_SENSOR_TYPE.TEMPERATURE, in_eSource := E_METIS_SENSOR_SOURCE.VOTER, in_nRampPeriodSec:= 10, in_lrFaultRamp:= 10);
t_sca_vot_7         (in_sName:='t_sca_vot_7',  in_eType := E_METIS_SENSOR_TYPE.TEMPERATURE, in_eSource := E_METIS_SENSOR_SOURCE.VOTER, in_nRampPeriodSec:= 10, in_lrFaultRamp:= 10);
t_sca_vot_8         (in_sName:='t_sca_vot_8',  in_eType := E_METIS_SENSOR_TYPE.TEMPERATURE, in_eSource := E_METIS_SENSOR_SOURCE.VOTER, in_nRampPeriodSec:= 10, in_lrFaultRamp:= 10);
t_sca_vot_9         (in_sName:='t_sca_vot_9',  in_eType := E_METIS_SENSOR_TYPE.TEMPERATURE, in_eSource := E_METIS_SENSOR_SOURCE.VOTER, in_nRampPeriodSec:= 10, in_lrFaultRamp:= 10);
t_sca_vot_10        (in_sName:='t_sca_vot_10', in_eType := E_METIS_SENSOR_TYPE.TEMPERATURE, in_eSource := E_METIS_SENSOR_SOURCE.VOTER, in_nRampPeriodSec:= 10, in_lrFaultRamp:= 10);
t_sca_wuh_ramp      (in_sName:='t_sca_wuh_ramp'  , in_eType := E_METIS_SENSOR_TYPE.TEMPERATURE, in_eSource := E_METIS_SENSOR_SOURCE.RAMP, in_nRampPeriodSec:= 10, in_lrFaultRamp:= 10);
t_sca_det_2_ramp    (in_sName:='t_sca_det_2_ramp', in_eType := E_METIS_SENSOR_TYPE.TEMPERATURE, in_eSource := E_METIS_SENSOR_SOURCE.RAMP, in_nRampPeriodSec:= 10, in_lrFaultRamp:= 10);
t_sca_dhs_2_ramp    (in_sName:='t_sca_dhs_2_ramp', in_eType := E_METIS_SENSOR_TYPE.TEMPERATURE, in_eSource := E_METIS_SENSOR_SOURCE.RAMP, in_nRampPeriodSec:= 10, in_lrFaultRamp:= 10);

(*IMG Temps*)       

t_img_lpw_1         (in_sName:='t_img_lpw_1', in_eType := E_METIS_SENSOR_TYPE.TEMPERATURE, in_eSource := E_METIS_SENSOR_SOURCE.LS240, in_nRampPeriodSec:= 10, in_lrFaultRamp:= 10);    
t_img_lpw_2         (in_sName:='t_img_lpw_2', in_eType := E_METIS_SENSOR_TYPE.TEMPERATURE, in_eSource := E_METIS_SENSOR_SOURCE.LS240, in_nRampPeriodSec:= 10, in_lrFaultRamp:= 10);    
t_img_lfw_1         (in_sName:='t_img_lfw_1', in_eType := E_METIS_SENSOR_TYPE.TEMPERATURE, in_eSource := E_METIS_SENSOR_SOURCE.LS240, in_nRampPeriodSec:= 10, in_lrFaultRamp:= 10);    
t_img_lfw_2         (in_sName:='t_img_lfw_2', in_eType := E_METIS_SENSOR_TYPE.TEMPERATURE, in_eSource := E_METIS_SENSOR_SOURCE.LS240, in_nRampPeriodSec:= 10, in_lrFaultRamp:= 10);    
t_img_lpr_1         (in_sName:='t_img_lpr_1', in_eType := E_METIS_SENSOR_TYPE.TEMPERATURE, in_eSource := E_METIS_SENSOR_SOURCE.LS240, in_nRampPeriodSec:= 10, in_lrFaultRamp:= 10);    
t_img_bwu_3         (in_sName:='t_img_bwu_3', in_eType := E_METIS_SENSOR_TYPE.TEMPERATURE, in_eSource := E_METIS_SENSOR_SOURCE.LS240, in_nRampPeriodSec:= 10, in_lrFaultRamp:= 10);    
t_img_lnd_1         (in_sName:='t_img_lnd_1', in_eType := E_METIS_SENSOR_TYPE.TEMPERATURE, in_eSource := E_METIS_SENSOR_SOURCE.LS240, in_nRampPeriodSec:= 10, in_lrFaultRamp:= 10);    
t_img_lnd_2         (in_sName:='t_img_lnd_2', in_eType := E_METIS_SENSOR_TYPE.TEMPERATURE, in_eSource := E_METIS_SENSOR_SOURCE.LS240, in_nRampPeriodSec:= 10, in_lrFaultRamp:= 10);    
t_img_npw_1         (in_sName:='t_img_npw_1', in_eType := E_METIS_SENSOR_TYPE.TEMPERATURE, in_eSource := E_METIS_SENSOR_SOURCE.LS240, in_nRampPeriodSec:= 10, in_lrFaultRamp:= 10);    
t_img_npw_2         (in_sName:='t_img_npw_2', in_eType := E_METIS_SENSOR_TYPE.TEMPERATURE, in_eSource := E_METIS_SENSOR_SOURCE.LS240, in_nRampPeriodSec:= 10, in_lrFaultRamp:= 10);    
t_img_nfw_1         (in_sName:='t_img_nfw_1', in_eType := E_METIS_SENSOR_TYPE.TEMPERATURE, in_eSource := E_METIS_SENSOR_SOURCE.LS240, in_nRampPeriodSec:= 10, in_lrFaultRamp:= 10);    
t_img_nfw_2         (in_sName:='t_img_nfw_2', in_eType := E_METIS_SENSOR_TYPE.TEMPERATURE, in_eSource := E_METIS_SENSOR_SOURCE.LS240, in_nRampPeriodSec:= 10, in_lrFaultRamp:= 10);    
t_img_npr_1         (in_sName:='t_img_npr_1', in_eType := E_METIS_SENSOR_TYPE.TEMPERATURE, in_eSource := E_METIS_SENSOR_SOURCE.LS240, in_nRampPeriodSec:= 10, in_lrFaultRamp:= 10);    
t_img_bwu_2         (in_sName:='t_img_bwu_2', in_eType := E_METIS_SENSOR_TYPE.TEMPERATURE, in_eSource := E_METIS_SENSOR_SOURCE.LS240, in_nRampPeriodSec:= 10, in_lrFaultRamp:= 10);    
t_img_nnd_1         (in_sName:='t_img_nnd_1', in_eType := E_METIS_SENSOR_TYPE.TEMPERATURE, in_eSource := E_METIS_SENSOR_SOURCE.LS240, in_nRampPeriodSec:= 10, in_lrFaultRamp:= 10);    
t_img_nnd_2         (in_sName:='t_img_nnd_2', in_eType := E_METIS_SENSOR_TYPE.TEMPERATURE, in_eSource := E_METIS_SENSOR_SOURCE.LS240, in_nRampPeriodSec:= 10, in_lrFaultRamp:= 10);    
t_img_opt_1         (in_sName:='t_img_opt_1', in_eType := E_METIS_SENSOR_TYPE.TEMPERATURE, in_eSource := E_METIS_SENSOR_SOURCE.LS240, in_nRampPeriodSec:= 10, in_lrFaultRamp:= 10);    
t_img_bwu_1         (in_sName:='t_img_bwu_1', in_eType := E_METIS_SENSOR_TYPE.TEMPERATURE, in_eSource := E_METIS_SENSOR_SOURCE.LS240, in_nRampPeriodSec:= 10, in_lrFaultRamp:= 10);    
t_img_ctr_1         (in_sName:='t_img_ctr_1', in_eType := E_METIS_SENSOR_TYPE.TEMPERATURE, in_eSource := E_METIS_SENSOR_SOURCE.LS240, in_nRampPeriodSec:= 10, in_lrFaultRamp:= 10);    
t_img_ctr_2         (in_sName:='t_img_ctr_2', in_eType := E_METIS_SENSOR_TYPE.TEMPERATURE, in_eSource := E_METIS_SENSOR_SOURCE.LS240, in_nRampPeriodSec:= 10, in_lrFaultRamp:= 10);    
t_img_70k_1         (in_sName:='t_img_70k_1', in_eType := E_METIS_SENSOR_TYPE.TEMPERATURE, in_eSource := E_METIS_SENSOR_SOURCE.LS240, in_nRampPeriodSec:= 10, in_lrFaultRamp:= 10);    
t_img_ln2_1         (in_sName:='t_img_ln2_1', in_eType := E_METIS_SENSOR_TYPE.TEMPERATURE, in_eSource := E_METIS_SENSOR_SOURCE.LS240, in_nRampPeriodSec:= 10, in_lrFaultRamp:= 10);    
t_img_ln2_2		    (in_sName:='t_img_ln2_2', in_eType := E_METIS_SENSOR_TYPE.TEMPERATURE, in_eSource := E_METIS_SENSOR_SOURCE.LS240, in_nRampPeriodSec:= 10, in_lrFaultRamp:= 10);	
t_img_hex_1         (in_sName:='t_img_hex_1', in_eType := E_METIS_SENSOR_TYPE.TEMPERATURE, in_eSource := E_METIS_SENSOR_SOURCE.LS240, in_nRampPeriodSec:= 10, in_lrFaultRamp:= 10);    
t_img_lmd_1         (in_sName:='t_img_lmd_1',  in_eType := E_METIS_SENSOR_TYPE.TEMPERATURE, in_eSource := E_METIS_SENSOR_SOURCE.LS336, in_nRampPeriodSec:= 10, in_lrFaultRamp:= 10);
t_img_lmd_2         (in_sName:='t_img_lmd_2',  in_eType := E_METIS_SENSOR_TYPE.TEMPERATURE, in_eSource := E_METIS_SENSOR_SOURCE.LS336, in_nRampPeriodSec:= 10, in_lrFaultRamp:= 10);
t_img_lmp_1         (in_sName:='t_img_lmp_1',  in_eType := E_METIS_SENSOR_TYPE.TEMPERATURE, in_eSource := E_METIS_SENSOR_SOURCE.LS336, in_nRampPeriodSec:= 10, in_lrFaultRamp:= 10);
t_img_lmp_2         (in_sName:='t_img_lmp_2',  in_eType := E_METIS_SENSOR_TYPE.TEMPERATURE, in_eSource := E_METIS_SENSOR_SOURCE.LS336, in_nRampPeriodSec:= 10, in_lrFaultRamp:= 10);
t_img_nd_1          (in_sName:='t_img_nd_1' ,  in_eType := E_METIS_SENSOR_TYPE.TEMPERATURE, in_eSource := E_METIS_SENSOR_SOURCE.LS336, in_nRampPeriodSec:= 10, in_lrFaultRamp:= 10);
t_img_nd_2          (in_sName:='t_img_nd_2' ,  in_eType := E_METIS_SENSOR_TYPE.TEMPERATURE, in_eSource := E_METIS_SENSOR_SOURCE.LS336, in_nRampPeriodSec:= 10, in_lrFaultRamp:= 10);
t_img_vot_1         (in_sName:='t_img_vot_1',  in_eType := E_METIS_SENSOR_TYPE.TEMPERATURE, in_eSource := E_METIS_SENSOR_SOURCE.VOTER, in_nRampPeriodSec:= 10, in_lrFaultRamp:= 10);
t_img_vot_2         (in_sName:='t_img_vot_2',  in_eType := E_METIS_SENSOR_TYPE.TEMPERATURE, in_eSource := E_METIS_SENSOR_SOURCE.VOTER, in_nRampPeriodSec:= 10, in_lrFaultRamp:= 10);
t_img_vot_3         (in_sName:='t_img_vot_3',  in_eType := E_METIS_SENSOR_TYPE.TEMPERATURE, in_eSource := E_METIS_SENSOR_SOURCE.VOTER, in_nRampPeriodSec:= 10, in_lrFaultRamp:= 10);
t_img_vot_4         (in_sName:='t_img_vot_4',  in_eType := E_METIS_SENSOR_TYPE.TEMPERATURE, in_eSource := E_METIS_SENSOR_SOURCE.VOTER, in_nRampPeriodSec:= 10, in_lrFaultRamp:= 10);
t_img_vot_5         (in_sName:='t_img_vot_5',  in_eType := E_METIS_SENSOR_TYPE.TEMPERATURE, in_eSource := E_METIS_SENSOR_SOURCE.VOTER, in_nRampPeriodSec:= 10, in_lrFaultRamp:= 10);
t_img_vot_6         (in_sName:='t_img_vot_6',  in_eType := E_METIS_SENSOR_TYPE.TEMPERATURE, in_eSource := E_METIS_SENSOR_SOURCE.VOTER, in_nRampPeriodSec:= 10, in_lrFaultRamp:= 10);
t_img_vot_7         (in_sName:='t_img_vot_7',  in_eType := E_METIS_SENSOR_TYPE.TEMPERATURE, in_eSource := E_METIS_SENSOR_SOURCE.VOTER, in_nRampPeriodSec:= 10, in_lrFaultRamp:= 10);
t_img_vot_8         (in_sName:='t_img_vot_8',  in_eType := E_METIS_SENSOR_TYPE.TEMPERATURE, in_eSource := E_METIS_SENSOR_SOURCE.VOTER, in_nRampPeriodSec:= 10, in_lrFaultRamp:= 10);
t_img_vot_9         (in_sName:='t_img_vot_9',  in_eType := E_METIS_SENSOR_TYPE.TEMPERATURE, in_eSource := E_METIS_SENSOR_SOURCE.VOTER, in_nRampPeriodSec:= 10, in_lrFaultRamp:= 10);
t_img_vot_10        (in_sName:='t_img_vot_10', in_eType := E_METIS_SENSOR_TYPE.TEMPERATURE, in_eSource := E_METIS_SENSOR_SOURCE.VOTER, in_nRampPeriodSec:= 10, in_lrFaultRamp:= 10);
t_img_wuh_ramp      (in_sName:='t_img_wuh_ramp'  , in_eType := E_METIS_SENSOR_TYPE.TEMPERATURE, in_eSource := E_METIS_SENSOR_SOURCE.RAMP, in_nRampPeriodSec:= 10, in_lrFaultRamp:= 10);
t_img_lmd_2_ramp    (in_sName:='t_img_lmd_2_ramp', in_eType := E_METIS_SENSOR_TYPE.TEMPERATURE, in_eSource := E_METIS_SENSOR_SOURCE.RAMP, in_nRampPeriodSec:= 10, in_lrFaultRamp:= 10);
t_img_lmp_2_ramp    (in_sName:='t_img_lmp_2_ramp', in_eType := E_METIS_SENSOR_TYPE.TEMPERATURE, in_eSource := E_METIS_SENSOR_SOURCE.RAMP, in_nRampPeriodSec:= 10, in_lrFaultRamp:= 10);
t_img_nd_2_ramp     (in_sName:='t_img_nd_2_ramp' , in_eType := E_METIS_SENSOR_TYPE.TEMPERATURE, in_eSource := E_METIS_SENSOR_SOURCE.RAMP, in_nRampPeriodSec:= 10, in_lrFaultRamp:= 10);

(*Temp LMS*)            
                        
t_lms_pma_1         (in_sName:='t_lms_pma_1', in_eType := E_METIS_SENSOR_TYPE.TEMPERATURE, in_eSource := E_METIS_SENSOR_SOURCE.LS240, in_nRampPeriodSec:= 10, in_lrFaultRamp:= 10);    
t_lms_pma_2         (in_sName:='t_lms_pma_2', in_eType := E_METIS_SENSOR_TYPE.TEMPERATURE, in_eSource := E_METIS_SENSOR_SOURCE.LS240, in_nRampPeriodSec:= 10, in_lrFaultRamp:= 10);    
t_lms_msa_1         (in_sName:='t_lms_msa_1', in_eType := E_METIS_SENSOR_TYPE.TEMPERATURE, in_eSource := E_METIS_SENSOR_SOURCE.LS240, in_nRampPeriodSec:= 10, in_lrFaultRamp:= 10);    
t_lms_msa_2         (in_sName:='t_lms_msa_2', in_eType := E_METIS_SENSOR_TYPE.TEMPERATURE, in_eSource := E_METIS_SENSOR_SOURCE.LS240, in_nRampPeriodSec:= 10, in_lrFaultRamp:= 10);    
t_lms_pra_1         (in_sName:='t_lms_pra_1', in_eType := E_METIS_SENSOR_TYPE.TEMPERATURE, in_eSource := E_METIS_SENSOR_SOURCE.LS240, in_nRampPeriodSec:= 10, in_lrFaultRamp:= 10);    
t_lms_pra_2         (in_sName:='t_lms_pra_2', in_eType := E_METIS_SENSOR_TYPE.TEMPERATURE, in_eSource := E_METIS_SENSOR_SOURCE.LS240, in_nRampPeriodSec:= 10, in_lrFaultRamp:= 10);    
t_lms_gra_1         (in_sName:='t_lms_gra_1', in_eType := E_METIS_SENSOR_TYPE.TEMPERATURE, in_eSource := E_METIS_SENSOR_SOURCE.LS240, in_nRampPeriodSec:= 10, in_lrFaultRamp:= 10);    
t_lms_gra_2         (in_sName:='t_lms_gra_2', in_eType := E_METIS_SENSOR_TYPE.TEMPERATURE, in_eSource := E_METIS_SENSOR_SOURCE.LS240, in_nRampPeriodSec:= 10, in_lrFaultRamp:= 10);    
t_lms_pla_1         (in_sName:='t_lms_pla_1', in_eType := E_METIS_SENSOR_TYPE.TEMPERATURE, in_eSource := E_METIS_SENSOR_SOURCE.LS240, in_nRampPeriodSec:= 10, in_lrFaultRamp:= 10);    
t_lms_pla_2         (in_sName:='t_lms_pla_2', in_eType := E_METIS_SENSOR_TYPE.TEMPERATURE, in_eSource := E_METIS_SENSOR_SOURCE.LS240, in_nRampPeriodSec:= 10, in_lrFaultRamp:= 10);    
t_lms_pla_3         (in_sName:='t_lms_pla_3', in_eType := E_METIS_SENSOR_TYPE.TEMPERATURE, in_eSource := E_METIS_SENSOR_SOURCE.LS240, in_nRampPeriodSec:= 10, in_lrFaultRamp:= 10);    
t_lms_pla_4         (in_sName:='t_lms_pla_4', in_eType := E_METIS_SENSOR_TYPE.TEMPERATURE, in_eSource := E_METIS_SENSOR_SOURCE.LS240, in_nRampPeriodSec:= 10, in_lrFaultRamp:= 10);    
t_lms_tma           (in_sName:='t_lms_tma',   in_eType := E_METIS_SENSOR_TYPE.TEMPERATURE, in_eSource := E_METIS_SENSOR_SOURCE.LS240, in_nRampPeriodSec:= 10, in_lrFaultRamp:= 10);    
t_lms_dtw           (in_sName:='t_lms_dtw',   in_eType := E_METIS_SENSOR_TYPE.TEMPERATURE, in_eSource := E_METIS_SENSOR_SOURCE.LS240, in_nRampPeriodSec:= 10, in_lrFaultRamp:= 10);    
t_lms_ptw           (in_sName:='t_lms_ptw',   in_eType := E_METIS_SENSOR_TYPE.TEMPERATURE, in_eSource := E_METIS_SENSOR_SOURCE.LS240, in_nRampPeriodSec:= 10, in_lrFaultRamp:= 10);    
t_lms_spare         (in_sName:='t_lms_spare', in_eType := E_METIS_SENSOR_TYPE.TEMPERATURE, in_eSource := E_METIS_SENSOR_SOURCE.LS240, in_nRampPeriodSec:= 10, in_lrFaultRamp:= 10);    
                      
(*Temp CFO*)

// Ambient sensors
t_cry_pca           (in_sName:='t_cry_pca', in_eType := E_METIS_SENSOR_TYPE.TEMPERATURE, in_eSource := E_METIS_SENSOR_SOURCE.EL32XX, in_lrScale := 0.01, in_lrOffset := 273.15);
t_cry_pcb           (in_sName:='t_cry_pcb', in_eType := E_METIS_SENSOR_TYPE.TEMPERATURE, in_eSource := E_METIS_SENSOR_SOURCE.EL32XX, in_lrScale := 0.01, in_lrOffset := 273.15);
t_cry_wim           (in_sName:='t_cry_wim', in_eType := E_METIS_SENSOR_TYPE.TEMPERATURE, in_eSource := E_METIS_SENSOR_SOURCE.EL32XX, in_lrScale := 0.01, in_lrOffset := 273.15);
t_cry_wia           (in_sName:='t_cry_wia', in_eType := E_METIS_SENSOR_TYPE.TEMPERATURE, in_eSource := E_METIS_SENSOR_SOURCE.EL32XX, in_lrScale := 0.01, in_lrOffset := 273.15);
// dew point calculation
t_cry_wid           (in_sName:='t_cry_wid', in_eType := E_METIS_SENSOR_TYPE.TEMPERATURE, in_eSource := E_METIS_SENSOR_SOURCE.DEW_POINT_CALC);

(*System temperatures   (3) *)
// Master temperature to estimate overall temperature of the cryostat  

t_master       		(in_sName:='t_master',  in_eType := E_METIS_SENSOR_TYPE.TEMPERATURE, in_eSource := E_METIS_SENSOR_SOURCE.VOTER, in_nRampPeriodSec:= 10, in_lrFaultRamp:= 10);
t_master_vot_1 		(in_sName:='t_master_vot_1',  in_eType := E_METIS_SENSOR_TYPE.TEMPERATURE, in_eSource := E_METIS_SENSOR_SOURCE.VOTER, in_nRampPeriodSec:= 10, in_lrFaultRamp:= 10);
t_master_vot_2 		(in_sName:='t_master_vot_2',  in_eType := E_METIS_SENSOR_TYPE.TEMPERATURE, in_eSource := E_METIS_SENSOR_SOURCE.VOTER, in_nRampPeriodSec:= 10, in_lrFaultRamp:= 10);
END_METHOD

METHOD M_SetTemperatureSensor : POINTER TO FB_METIS_TEMPERATURE
VAR_INPUT
	m_nIndex	:	INT;
END_VAR
// always return a valid pointer!
IF (m_nIndex >= MIN_INDEX) AND (m_nIndex <= MAX_INDEX) THEN 
    M_SetTemperatureSensor := all_temperatures[m_nIndex];
ELSE
    M_SetTemperatureSensor := all_temperatures[0]; // empty temperature
END_IF
END_METHOD

METHOD M_UpdatePointer
VAR_INPUT
    pSensor : POINTER TO FB_METIS_TEMPERATURE;
END_VAR
VAR_IN_OUT
    i : INT;
END_VAR
IF i >= MIN_INDEX AND i <= MAX_INDEX THEN
    all_temperatures[i] := pSensor;
    i := i + 1;
END_IF
END_METHOD

METHOD M_UpdatePointers
VAR_INPUT
END_VAR
VAR_INST
    {attribute 'OPC.UA.DA' := '0'}
    i : INT := 0;
END_VAR
// EMPTY
M_UpdatePointer(i := i, pSensor := ADR(empty_temp));

// CRY
M_UpdatePointer(i := i, pSensor := ADR(t_cry_sha_1));
M_UpdatePointer(i := i, pSensor := ADR(t_cry_sha_2));
M_UpdatePointer(i := i, pSensor := ADR(t_cry_sha_3));
M_UpdatePointer(i := i, pSensor := ADR(t_cry_sha_4));
M_UpdatePointer(i := i, pSensor := ADR(t_cry_shb_1));
M_UpdatePointer(i := i, pSensor := ADR(t_cry_shb_2));
M_UpdatePointer(i := i, pSensor := ADR(t_cry_shb_3));
M_UpdatePointer(i := i, pSensor := ADR(t_cry_shb_4));
M_UpdatePointer(i := i, pSensor := ADR(t_cry_shc_1));
M_UpdatePointer(i := i, pSensor := ADR(t_cry_shc_2));
M_UpdatePointer(i := i, pSensor := ADR(t_cry_shc_3));
M_UpdatePointer(i := i, pSensor := ADR(t_cry_shc_4));
M_UpdatePointer(i := i, pSensor := ADR(t_cry_pta_1));
M_UpdatePointer(i := i, pSensor := ADR(t_cry_pta_2));
M_UpdatePointer(i := i, pSensor := ADR(t_cry_ptb_1));
M_UpdatePointer(i := i, pSensor := ADR(t_cry_ptb_2));
M_UpdatePointer(i := i, pSensor := ADR(t_cry_ptc_1));
M_UpdatePointer(i := i, pSensor := ADR(t_cry_ptc_2));
M_UpdatePointer(i := i, pSensor := ADR(t_cry_pta_3));
M_UpdatePointer(i := i, pSensor := ADR(t_cry_ptb_3));
M_UpdatePointer(i := i, pSensor := ADR(t_cry_ptc_3));
M_UpdatePointer(i := i, pSensor := ADR(t_cry_sp_1));
M_UpdatePointer(i := i, pSensor := ADR(t_cry_sp_2));
M_UpdatePointer(i := i, pSensor := ADR(t_cry_vot_1));
M_UpdatePointer(i := i, pSensor := ADR(t_cry_vot_2));
M_UpdatePointer(i := i, pSensor := ADR(t_cry_vot_3));
M_UpdatePointer(i := i, pSensor := ADR(t_cry_vot_4));
M_UpdatePointer(i := i, pSensor := ADR(t_cry_vot_5));
M_UpdatePointer(i := i, pSensor := ADR(t_cry_vot_6));
M_UpdatePointer(i := i, pSensor := ADR(t_cry_vot_7));
M_UpdatePointer(i := i, pSensor := ADR(t_cry_vot_8));
M_UpdatePointer(i := i, pSensor := ADR(t_cry_vot_9));
M_UpdatePointer(i := i, pSensor := ADR(t_cry_vot_10));

// SCA
M_UpdatePointer(i := i, pSensor := ADR(t_sca_fw_1));
M_UpdatePointer(i := i, pSensor := ADR(t_sca_fw_2));
M_UpdatePointer(i := i, pSensor := ADR(t_sca_lu_1));
M_UpdatePointer(i := i, pSensor := ADR(t_sca_fm));
M_UpdatePointer(i := i, pSensor := ADR(t_sca_fs));
M_UpdatePointer(i := i, pSensor := ADR(t_sca_lu_2));
M_UpdatePointer(i := i, pSensor := ADR(t_sca_mod));
M_UpdatePointer(i := i, pSensor := ADR(t_sca_pyr));
M_UpdatePointer(i := i, pSensor := ADR(t_sca_h_1));
M_UpdatePointer(i := i, pSensor := ADR(t_sca_if_1));
M_UpdatePointer(i := i, pSensor := ADR(t_sca_if_2));
M_UpdatePointer(i := i, pSensor := ADR(t_sca_lu_3));
M_UpdatePointer(i := i, pSensor := ADR(t_sca_bp_1));
M_UpdatePointer(i := i, pSensor := ADR(t_sca_bp_2));
M_UpdatePointer(i := i, pSensor := ADR(t_sca_bp_3));
M_UpdatePointer(i := i, pSensor := ADR(t_sca_h_2));
M_UpdatePointer(i := i, pSensor := ADR(t_sca_det_1));
M_UpdatePointer(i := i, pSensor := ADR(t_sca_det_2));
M_UpdatePointer(i := i, pSensor := ADR(t_sca_dhs_1));
M_UpdatePointer(i := i, pSensor := ADR(t_sca_dhs_2));
M_UpdatePointer(i := i, pSensor := ADR(t_sca_vot_1));
M_UpdatePointer(i := i, pSensor := ADR(t_sca_vot_2));
M_UpdatePointer(i := i, pSensor := ADR(t_sca_vot_3));
M_UpdatePointer(i := i, pSensor := ADR(t_sca_vot_4));
M_UpdatePointer(i := i, pSensor := ADR(t_sca_vot_5));
M_UpdatePointer(i := i, pSensor := ADR(t_sca_vot_6));
M_UpdatePointer(i := i, pSensor := ADR(t_sca_vot_7));
M_UpdatePointer(i := i, pSensor := ADR(t_sca_vot_8));
M_UpdatePointer(i := i, pSensor := ADR(t_sca_vot_9));
M_UpdatePointer(i := i, pSensor := ADR(t_sca_vot_10));
M_UpdatePointer(i := i, pSensor := ADR(t_sca_wuh_ramp));
M_UpdatePointer(i := i, pSensor := ADR(t_sca_det_2_ramp));
M_UpdatePointer(i := i, pSensor := ADR(t_sca_dhs_2_ramp));

// IMG
M_UpdatePointer(i := i, pSensor := ADR(t_img_lpw_1));
M_UpdatePointer(i := i, pSensor := ADR(t_img_lpw_2));
M_UpdatePointer(i := i, pSensor := ADR(t_img_lfw_1));
M_UpdatePointer(i := i, pSensor := ADR(t_img_lfw_2));
M_UpdatePointer(i := i, pSensor := ADR(t_img_lpr_1));
M_UpdatePointer(i := i, pSensor := ADR(t_img_bwu_3));
M_UpdatePointer(i := i, pSensor := ADR(t_img_lnd_1));
M_UpdatePointer(i := i, pSensor := ADR(t_img_lnd_2));
M_UpdatePointer(i := i, pSensor := ADR(t_img_npw_1));
M_UpdatePointer(i := i, pSensor := ADR(t_img_npw_2));
M_UpdatePointer(i := i, pSensor := ADR(t_img_nfw_1));
M_UpdatePointer(i := i, pSensor := ADR(t_img_nfw_2));
M_UpdatePointer(i := i, pSensor := ADR(t_img_npr_1));
M_UpdatePointer(i := i, pSensor := ADR(t_img_bwu_2));
M_UpdatePointer(i := i, pSensor := ADR(t_img_nnd_1));
M_UpdatePointer(i := i, pSensor := ADR(t_img_nnd_2));
M_UpdatePointer(i := i, pSensor := ADR(t_img_opt_1));
M_UpdatePointer(i := i, pSensor := ADR(t_img_bwu_1));
M_UpdatePointer(i := i, pSensor := ADR(t_img_ctr_1));
M_UpdatePointer(i := i, pSensor := ADR(t_img_ctr_2));
M_UpdatePointer(i := i, pSensor := ADR(t_img_70k_1));
M_UpdatePointer(i := i, pSensor := ADR(t_img_ln2_1));
M_UpdatePointer(i := i, pSensor := ADR(t_img_ln2_2));
M_UpdatePointer(i := i, pSensor := ADR(t_img_hex_1));
M_UpdatePointer(i := i, pSensor := ADR(t_img_lmd_1));
M_UpdatePointer(i := i, pSensor := ADR(t_img_lmd_2));
M_UpdatePointer(i := i, pSensor := ADR(t_img_lmp_1));
M_UpdatePointer(i := i, pSensor := ADR(t_img_lmp_2));
M_UpdatePointer(i := i, pSensor := ADR(t_img_nd_1));
M_UpdatePointer(i := i, pSensor := ADR(t_img_nd_2));
M_UpdatePointer(i := i, pSensor := ADR(t_img_vot_1));
M_UpdatePointer(i := i, pSensor := ADR(t_img_vot_2));
M_UpdatePointer(i := i, pSensor := ADR(t_img_vot_3));
M_UpdatePointer(i := i, pSensor := ADR(t_img_vot_4));
M_UpdatePointer(i := i, pSensor := ADR(t_img_vot_5));
M_UpdatePointer(i := i, pSensor := ADR(t_img_vot_6));
M_UpdatePointer(i := i, pSensor := ADR(t_img_vot_7));
M_UpdatePointer(i := i, pSensor := ADR(t_img_vot_8));
M_UpdatePointer(i := i, pSensor := ADR(t_img_vot_9));
M_UpdatePointer(i := i, pSensor := ADR(t_img_vot_10));
M_UpdatePointer(i := i, pSensor := ADR(t_img_wuh_ramp));
M_UpdatePointer(i := i, pSensor := ADR(t_img_lmd_2_ramp));
M_UpdatePointer(i := i, pSensor := ADR(t_img_lmp_2_ramp));
M_UpdatePointer(i := i, pSensor := ADR(t_img_nd_2_ramp));

// LMS
M_UpdatePointer(i := i, pSensor := ADR(t_lms_pma_1));
M_UpdatePointer(i := i, pSensor := ADR(t_lms_pma_2));
M_UpdatePointer(i := i, pSensor := ADR(t_lms_msa_1));
M_UpdatePointer(i := i, pSensor := ADR(t_lms_msa_2));
M_UpdatePointer(i := i, pSensor := ADR(t_lms_pra_1));
M_UpdatePointer(i := i, pSensor := ADR(t_lms_pra_2));
M_UpdatePointer(i := i, pSensor := ADR(t_lms_gra_1));
M_UpdatePointer(i := i, pSensor := ADR(t_lms_gra_2));
M_UpdatePointer(i := i, pSensor := ADR(t_lms_pla_1));
M_UpdatePointer(i := i, pSensor := ADR(t_lms_pla_2));
M_UpdatePointer(i := i, pSensor := ADR(t_lms_pla_3));
M_UpdatePointer(i := i, pSensor := ADR(t_lms_pla_4));
M_UpdatePointer(i := i, pSensor := ADR(t_lms_tma));
M_UpdatePointer(i := i, pSensor := ADR(t_lms_dtw));
M_UpdatePointer(i := i, pSensor := ADR(t_lms_ptw));
M_UpdatePointer(i := i, pSensor := ADR(t_lms_spare));

// Ambient
M_UpdatePointer(i := i, pSensor := ADR(t_cry_pca));
M_UpdatePointer(i := i, pSensor := ADR(t_cry_pcb));
M_UpdatePointer(i := i, pSensor := ADR(t_cry_wim));
M_UpdatePointer(i := i, pSensor := ADR(t_cry_wia));
M_UpdatePointer(i := i, pSensor := ADR(t_cry_wid));

(*System temperatures   (3) *)
M_UpdatePointer(i := i, pSensor := ADR(t_master));
M_UpdatePointer(i := i, pSensor := ADR(t_master_vot_1));
M_UpdatePointer(i := i, pSensor := ADR(t_master_vot_2));
END_METHOD

END_FUNCTION_BLOCK

// POUs/Devices/Temperature/FB_METIS_TEMPERATURE
FUNCTION_BLOCK FB_METIS_TEMPERATURE EXTENDS FB_METIS_SENSOR_BASE
VAR_INPUT
END_VAR
VAR_OUTPUT
END_VAR
VAR
    {attribute 'OPC.UA.DA' := '1'}
	{attribute 'TcHmiSymbol.ShowRecursively'}
    stat : T_METIS_TEMPERATURE_STATUS;
END_VAR

// update the references
RefStatBase Ref= stat;
RefStat Ref= stat;

SUPER^();

stat.lrTempK := stat.lrBaseValue;
stat.lrTempC := stat.lrTempK - 273.15;

END_FUNCTION_BLOCK

// POUs/Devices/Base_Sensor/FB_METIS_SENSOR_BASE
FUNCTION_BLOCK FB_METIS_SENSOR_BASE EXTENDS FB_CRYO_SENSOR_BASE
VAR_INPUT
	{attribute 'OPC.UA.DA' := '0'}
	in_eType:               E_METIS_SENSOR_TYPE;
	{attribute 'OPC.UA.DA' := '0'}
	in_eSource:             E_METIS_SENSOR_SOURCE;
	{attribute 'OPC.UA.DA' := '0'}
	in_nRampPeriodSec:		UDINT := 60;		// Ramp measurement period [sec]. Default 60 sec.
	{attribute 'OPC.UA.DA' := '0'}
	in_lrFaultRamp:			LREAL := 35;		// Ramp > in_nFaultRamp OR Ramp < -in_nFaultRamp(deg/min) indicate DT670 sensor fault.	

	{attribute 'OPC.UA.DA' := '0'}
    in_lrScale:             LREAL := 1.0;       // base value = input value x scale + offset
    {attribute 'OPC.UA.DA' := '0'}
    in_lrOffset:            LREAL := 0.0;       // offset value for EL32XX
    
    
